LIN {X 0,Y 487.922,Z 777.858,A -85,B 0,C 180,E1 -6674.706,E2 -6674.706} C_VEL
LIN {X 0,Y 487.963,Z 774.749,A -85,B 0,C 180,E1 -6677.604,E2 -6677.604} C_VEL
LIN {X 0,Y 487.996,Z 771.009,A -85,B 0,C 180,E1 -6681.102,E2 -6681.102} C_VEL
LIN {X 0,Y 488.063,Z 768.175,A -85,B 0,C 180,E1 -6683.777,E2 -6683.777} C_VEL
LIN {X 0,Y 488.138,Z 765.028,A -85,B 0,C 180,E1 -6686.791,E2 -6686.791} C_VEL
LIN {X 0,Y 488.198,Z 761.474,A -85,B 0,C 180,E1 -6690.259,E2 -6690.259} C_VEL
LIN {X 0,Y 488.191,Z 760.678,A -85,B 0,C 180,E1 -6691.214,E2 -6691.214} C_VEL
LIN {X 0,Y 488.524,Z 760.636,A -85,B 0,C 180,E1 -6694.128,E2 -6694.128} C_VEL
LIN {X 0,Y 488.663,Z 760.617,A -85,B 0,C 180,E1 -6697.159,E2 -6697.159} C_VEL
LIN {X 0,Y 488.714,Z 760.606,A -85,B 0,C 180,E1 -6700.344,E2 -6700.344} C_VEL
LIN {X 0,Y 488.682,Z 760.613,A -85,B 0,C 180,E1 -6703.653,E2 -6703.653} C_VEL
LIN {X 0,Y 488.682,Z 760.609,A -85,B 0,C 180,E1 -6706.345,E2 -6706.345} C_VEL
LIN {X 0,Y 488.727,Z 760.607,A -85,B 0,C 180,E1 -6709.676,E2 -6709.676} C_VEL
LIN {X 0,Y 488.672,Z 760.612,A -85,B 0,C 180,E1 -6712.84,E2 -6712.84} C_VEL
LIN {X 0,Y 488.716,Z 760.608,A -85,B 0,C 180,E1 -6715.886,E2 -6715.886} C_VEL
LIN {X 0,Y 488.683,Z 760.609,A -85,B 0,C 180,E1 -6718.819,E2 -6718.819} C_VEL
LIN {X 0,Y 488.691,Z 760.607,A -85,B 0,C 180,E1 -6720.347,E2 -6720.347} C_VEL
LIN {X 0,Y 488.027,Z 760.693,A -85,B 0,C 180,E1 -6721.035,E2 -6721.035} C_VEL
LIN {X 0,Y 485.161,Z 761.049,A -85,B 0,C 180,E1 -6722.153,E2 -6722.153} C_VEL
LIN {X 0,Y 482.747,Z 761.35,A -85,B 0,C 180,E1 -6723.053,E2 -6723.053} C_VEL
LIN {X 0,Y 481.727,Z 761.48,A -85,B 0,C 180,E1 -6723.749,E2 -6723.749} C_VEL
LIN {X 0,Y 481.654,Z 761.487,A -85,B 0,C 180,E1 -6723.985,E2 -6723.985} C_VEL
LIN {X 0,Y 481.665,Z 761.483,A -85,B 0,C 180,E1 -6726.811,E2 -6726.811} C_VEL
LIN {X 0,Y 481.686,Z 761.486,A -85,B 0,C 180,E1 -6729.502,E2 -6729.502} C_VEL
LIN {X 0,Y 481.679,Z 761.484,A -85,B 0,C 180,E1 -6732.157,E2 -6732.157} C_VEL
LIN {X 0,Y 481.732,Z 761.474,A -85,B 0,C 180,E1 -6734.775,E2 -6734.775} C_VEL
LIN {X 0,Y 481.74,Z 761.476,A -85,B 0,C 180,E1 -6738.215,E2 -6738.215} C_VEL
LIN {X 0,Y 481.709,Z 761.481,A -85,B 0,C 180,E1 -6741.611,E2 -6741.611} C_VEL
LIN {X 0,Y 481.763,Z 761.475,A -85,B 0,C 180,E1 -6744.139,E2 -6744.139} C_VEL
LIN {X 0,Y 481.895,Z 761.455,A -85,B 0,C 180,E1 -6747.492,E2 -6747.492} C_VEL
LIN {X 0,Y 481.899,Z 761.461,A -85,B 0,C 180,E1 -6750,E2 -6750} C_VEL
LIN {X 0,Y 481.893,Z 761.456,A -85,B 0,C 180,E1 -6752.508,E2 -6752.508} C_VEL
LIN {X 0,Y 481.76,Z 761.474,A -85,B 0,C 180,E1 -6755.861,E2 -6755.861} C_VEL
LIN {X 0,Y 481.701,Z 761.483,A -85,B 0,C 180,E1 -6758.389,E2 -6758.389} C_VEL
LIN {X 0,Y 481.724,Z 761.477,A -85,B 0,C 180,E1 -6761.786,E2 -6761.786} C_VEL
LIN {X 0,Y 481.732,Z 761.474,A -85,B 0,C 180,E1 -6765.225,E2 -6765.225} C_VEL
LIN {X 0,Y 481.696,Z 761.482,A -85,B 0,C 180,E1 -6768.722,E2 -6768.722} C_VEL
LIN {X 0,Y 481.636,Z 761.486,A -85,B 0,C 180,E1 -6771.395,E2 -6771.395} C_VEL
LIN {X 0,Y 481.639,Z 761.489,A -85,B 0,C 180,E1 -6774.115,E2 -6774.115} C_VEL
LIN {X 0,Y 481.667,Z 761.483,A -85,B 0,C 180,E1 -6777.123,E2 -6777.123} C_VEL
LIN {X 0,Y 481.664,Z 761.483,A -85,B 0,C 180,E1 -6779.742,E2 -6779.742} C_VEL
LIN {X 0,Y 481.662,Z 761.49,A -85,B 0,C 180,E1 -6782.675,E2 -6782.675} C_VEL
LIN {X 0,Y 481.628,Z 761.488,A -85,B 0,C 180,E1 -6785.71,E2 -6785.71} C_VEL
LIN {X 0,Y 481.664,Z 761.489,A -85,B 0,C 180,E1 -6788.86,E2 -6788.86} C_VEL
LIN {X 0,Y 481.646,Z 761.486,A -85,B 0,C 180,E1 -6791.914,E2 -6791.914} C_VEL
LIN {X 0,Y 481.649,Z 761.489,A -85,B 0,C 180,E1 -6794.459,E2 -6794.459} C_VEL
LIN {X 0,Y 481.643,Z 761.486,A -85,B 0,C 180,E1 -6797.84,E2 -6797.84} C_VEL
LIN {X 0,Y 481.676,Z 761.486,A -85,B 0,C 180,E1 -6800.652,E2 -6800.652} C_VEL
LIN {X 0,Y 481.618,Z 761.492,A -85,B 0,C 180,E1 -6803.378,E2 -6803.378} C_VEL
LIN {X 0,Y 481.486,Z 761.51,A -85,B 0,C 180,E1 -6806.314,E2 -6806.314} C_VEL
LIN {X 0,Y 481.112,Z 761.559,A -85,B 0,C 180,E1 -6809.253,E2 -6809.253} C_VEL
LIN {X 0,Y 480.968,Z 761.685,A -85,B 0,C 180,E1 -6810.212,E2 -6810.212} C_VEL
LIN {X 0,Y 481.03,Z 764.86,A -85,B 0,C 180,E1 -6813.07,E2 -6813.07} C_VEL
LIN {X 0,Y 480.937,Z 767.926,A -85,B 0,C 180,E1 -6815.849,E2 -6815.849} C_VEL
LIN {X 0,Y 480.903,Z 770.923,A -85,B 0,C 180,E1 -6818.572,E2 -6818.572} C_VEL
LIN {X 0,Y 480.857,Z 773.831,A -85,B 0,C 180,E1 -6821.245,E2 -6821.245} C_VEL
LIN {X 0,Y 480.874,Z 777.672,A -85,B 0,C 180,E1 -6824.749,E2 -6824.749} C_VEL
LIN {X 0,Y 480.881,Z 778.156,A -85,B 0,C 180,E1 -6825.194,E2 -6825.194} C_VEL
LIN {X 0,Y 483.342,Z 790.593,A -85,B 0,C 180,E1 -6825.636,E2 -6825.636} C_VEL
LIN {X 0,Y 483.812,Z 796.114,A -85,B 0,C 180,E1 -6825.865,E2 -6825.865} C_VEL
LIN {X 0,Y 483.429,Z 808.116,A -85,B 0,C 180,E1 -6826.443,E2 -6826.443} C_VEL
LIN {X 0,Y 483.005,Z 820.229,A -85,B 0,C 180,E1 -6827.21,E2 -6827.21} C_VEL
LIN {X 0,Y 482.616,Z 831.531,A -85,B 0,C 180,E1 -6828.131,E2 -6828.131} C_VEL
LIN {X 0,Y 482.137,Z 840.94,A -85,B 0,C 180,E1 -6829.077,E2 -6829.077} C_VEL
LIN {X 0,Y 481.85,Z 849.541,A -85,B 0,C 180,E1 -6830.133,E2 -6830.133} C_VEL
LIN {X 0,Y 481.489,Z 857.935,A -85,B 0,C 180,E1 -6831.396,E2 -6831.396} C_VEL
LIN {X 0,Y 481.234,Z 863.639,A -85,B 0,C 180,E1 -6832.448,E2 -6832.448} C_VEL
LIN {X 0,Y 481.106,Z 869.017,A -85,B 0,C 180,E1 -6833.666,E2 -6833.666} C_VEL
LIN {X 0,Y 480.907,Z 873.547,A -85,B 0,C 180,E1 -6834.971,E2 -6834.971} C_VEL
LIN {X 0,Y 480.941,Z 875.835,A -85,B 0,C 180,E1 -6835.811,E2 -6835.811} C_VEL
LIN {X 0,Y 480.897,Z 877.707,A -85,B 0,C 180,E1 -6836.65,E2 -6836.65} C_VEL
LIN {X 0,Y 480.845,Z 879.143,A -85,B 0,C 180,E1 -6837.488,E2 -6837.488} C_VEL
LIN {X 0,Y 480.76,Z 880.779,A -85,B 0,C 180,E1 -6839.163,E2 -6839.163} C_VEL
LIN {X 0,Y 480.743,Z 881.028,A -85,B 0,C 180,E1 -6840.001,E2 -6840.001} C_VEL
LIN {X 0,Y 480.76,Z 880.847,A -85,B 0,C 180,E1 -6840.838,E2 -6840.838} C_VEL
LIN {X 0,Y 480.862,Z 879.314,A -85,B 0,C 180,E1 -6842.514,E2 -6842.514} C_VEL
LIN {X 0,Y 480.897,Z 877.961,A -85,B 0,C 180,E1 -6843.352,E2 -6843.352} C_VEL
LIN {X 0,Y 480.95,Z 875.11,A -85,B 0,C 180,E1 -6844.611,E2 -6844.611} C_VEL
LIN {X 0,Y 481.088,Z 871.224,A -85,B 0,C 180,E1 -6845.87,E2 -6845.87} C_VEL
LIN {X 0,Y 481.187,Z 866.185,A -85,B 0,C 180,E1 -6847.132,E2 -6847.132} C_VEL
LIN {X 0,Y 481.437,Z 859.82,A -85,B 0,C 180,E1 -6848.395,E2 -6848.395} C_VEL
LIN {X 0,Y 481.759,Z 851.905,A -85,B 0,C 180,E1 -6849.659,E2 -6849.659} C_VEL
LIN {X 0,Y 482.071,Z 843.809,A -85,B 0,C 180,E1 -6850.713,E2 -6850.713} C_VEL
LIN {X 0,Y 482.589,Z 833.83,A -85,B 0,C 180,E1 -6851.765,E2 -6851.765} C_VEL
LIN {X 0,Y 482.906,Z 822.414,A -85,B 0,C 180,E1 -6852.736,E2 -6852.736} C_VEL
LIN {X 0,Y 483.366,Z 811.702,A -85,B 0,C 180,E1 -6853.453,E2 -6853.453} C_VEL
LIN {X 0,Y 483.766,Z 799.439,A -85,B 0,C 180,E1 -6854.084,E2 -6854.084} C_VEL
LIN {X 0,Y 483.682,Z 793.011,A -85,B 0,C 180,E1 -6854.355,E2 -6854.355} C_VEL
LIN {X 0,Y 481.87,Z 782.956,A -85,B 0,C 180,E1 -6854.74,E2 -6854.74} C_VEL
LIN {X 0,Y 480.939,Z 778.913,A -85,B 0,C 180,E1 -6854.899,E2 -6854.899} C_VEL
LIN {X 0,Y 480.94,Z 775.326,A -85,B 0,C 180,E1 -6858.222,E2 -6858.222} C_VEL
LIN {X 0,Y 480.955,Z 771.748,A -85,B 0,C 180,E1 -6861.428,E2 -6861.428} C_VEL
LIN {X 0,Y 480.98,Z 768.696,A -85,B 0,C 180,E1 -6864.151,E2 -6864.151} C_VEL
LIN {X 0,Y 481.015,Z 765.283,A -85,B 0,C 180,E1 -6866.968,E2 -6866.968} C_VEL
LIN {X 0,Y 480.974,Z 761.647,A -85,B 0,C 180,E1 -6869.79,E2 -6869.79} C_VEL
LIN {X 0,Y 481.36,Z 761.528,A -85,B 0,C 180,E1 -6872.699,E2 -6872.699} C_VEL
LIN {X 0,Y 481.595,Z 761.495,A -85,B 0,C 180,E1 -6875.714,E2 -6875.714} C_VEL
LIN {X 0,Y 481.675,Z 761.487,A -85,B 0,C 180,E1 -6878.859,E2 -6878.859} C_VEL
LIN {X 0,Y 481.651,Z 761.486,A -85,B 0,C 180,E1 -6881.912,E2 -6881.912} C_VEL
LIN {X 0,Y 481.664,Z 761.486,A -85,B 0,C 180,E1 -6884.458,E2 -6884.458} C_VEL
LIN {X 0,Y 481.652,Z 761.487,A -85,B 0,C 180,E1 -6887.84,E2 -6887.84} C_VEL
LIN {X 0,Y 481.701,Z 761.516,A -85,B 0,C 180,E1 -6889.801,E2 -6889.801} C_VEL
LIN {X 0,Y 482.913,Z 768.412,A -85,B 0,C 180,E1 -6892.774,E2 -6892.774} C_VEL
LIN {X 0,Y 483.335,Z 772.686,A -85,B 0,C 180,E1 -6894.517,E2 -6894.517} C_VEL
LIN {X 0,Y 482.962,Z 780.236,A -85,B 0,C 180,E1 -6897.424,E2 -6897.424} C_VEL
LIN {X 0,Y 482.594,Z 788.032,A -85,B 0,C 180,E1 -6900.321,E2 -6900.321} C_VEL
LIN {X 0,Y 482.239,Z 795.887,A -85,B 0,C 180,E1 -6903.142,E2 -6903.142} C_VEL
LIN {X 0,Y 481.961,Z 803.794,A -85,B 0,C 180,E1 -6905.902,E2 -6905.902} C_VEL
LIN {X 0,Y 481.677,Z 813.021,A -85,B 0,C 180,E1 -6909.037,E2 -6909.037} C_VEL
LIN {X 0,Y 481.429,Z 822.408,A -85,B 0,C 180,E1 -6912.148,E2 -6912.148} C_VEL
LIN {X 0,Y 481.282,Z 831.603,A -85,B 0,C 180,E1 -6915.072,E2 -6915.072} C_VEL
LIN {X 0,Y 483.425,Z 845.293,A -85,B 0,C 180,E1 -6915.49,E2 -6915.49} C_VEL
LIN {X 0,Y 483.816,Z 849.512,A -85,B 0,C 180,E1 -6915.649,E2 -6915.649} C_VEL
LIN {X 0,Y 483.512,Z 861.696,A -85,B 0,C 180,E1 -6916.177,E2 -6916.177} C_VEL
LIN {X 0,Y 483.027,Z 873.992,A -85,B 0,C 180,E1 -6916.891,E2 -6916.891} C_VEL
LIN {X 0,Y 482.617,Z 884.929,A -85,B 0,C 180,E1 -6917.703,E2 -6917.703} C_VEL
LIN {X 0,Y 482.23,Z 895.247,A -85,B 0,C 180,E1 -6918.653,E2 -6918.653} C_VEL
LIN {X 0,Y 481.821,Z 904.529,A -85,B 0,C 180,E1 -6919.707,E2 -6919.707} C_VEL
LIN {X 0,Y 481.453,Z 913.564,A -85,B 0,C 180,E1 -6920.972,E2 -6920.972} C_VEL
LIN {X 0,Y 481.18,Z 920.842,A -85,B 0,C 180,E1 -6922.235,E2 -6922.235} C_VEL
LIN {X 0,Y 481.025,Z 926.557,A -85,B 0,C 180,E1 -6923.473,E2 -6923.473} C_VEL
LIN {X 0,Y 480.979,Z 930.536,A -85,B 0,C 180,E1 -6924.55,E2 -6924.55} C_VEL
LIN {X 0,Y 480.85,Z 934.181,A -85,B 0,C 180,E1 -6925.809,E2 -6925.809} C_VEL
LIN {X 0,Y 480.892,Z 936.066,A -85,B 0,C 180,E1 -6926.649,E2 -6926.649} C_VEL
LIN {X 0,Y 480.819,Z 938.478,A -85,B 0,C 180,E1 -6928.325,E2 -6928.325} C_VEL
LIN {X 0,Y 480.76,Z 939.086,A -85,B 0,C 180,E1 -6929.162,E2 -6929.162} C_VEL
LIN {X 0,Y 480.743,Z 939.297,A -85,B 0,C 180,E1 -6930,E2 -6930} C_VEL
LIN {X 0,Y 480.819,Z 938.457,A -85,B 0,C 180,E1 -6931.675,E2 -6931.675} C_VEL
LIN {X 0,Y 480.804,Z 937.443,A -85,B 0,C 180,E1 -6932.513,E2 -6932.513} C_VEL
LIN {X 0,Y 480.892,Z 936.018,A -85,B 0,C 180,E1 -6933.351,E2 -6933.351} C_VEL
LIN {X 0,Y 480.854,Z 933.023,A -85,B 0,C 180,E1 -6934.611,E2 -6934.611} C_VEL
LIN {X 0,Y 481.003,Z 928.98,A -85,B 0,C 180,E1 -6935.87,E2 -6935.87} C_VEL
LIN {X 0,Y 481.115,Z 922.75,A -85,B 0,C 180,E1 -6937.344,E2 -6937.344} C_VEL
LIN {X 0,Y 481.368,Z 915.951,A -85,B 0,C 180,E1 -6938.607,E2 -6938.607} C_VEL
LIN {X 0,Y 481.668,Z 907.498,A -85,B 0,C 180,E1 -6939.872,E2 -6939.872} C_VEL
LIN {X 0,Y 481.993,Z 898.816,A -85,B 0,C 180,E1 -6940.927,E2 -6940.927} C_VEL
LIN {X 0,Y 482.463,Z 888.126,A -85,B 0,C 180,E1 -6941.981,E2 -6941.981} C_VEL
LIN {X 0,Y 482.864,Z 876.533,A -85,B 0,C 180,E1 -6942.899,E2 -6942.899} C_VEL
LIN {X 0,Y 483.32,Z 863.934,A -85,B 0,C 180,E1 -6943.668,E2 -6943.668} C_VEL
LIN {X 0,Y 483.741,Z 851.423,A -85,B 0,C 180,E1 -6944.245,E2 -6944.245} C_VEL
LIN {X 0,Y 483.593,Z 846.689,A -85,B 0,C 180,E1 -6944.424,E2 -6944.424} C_VEL
LIN {X 0,Y 481.609,Z 833.971,A -85,B 0,C 180,E1 -6944.846,E2 -6944.846} C_VEL
LIN {X 0,Y 481.222,Z 830.609,A -85,B 0,C 180,E1 -6944.943,E2 -6944.943} C_VEL
LIN {X 0,Y 481.439,Z 819.625,A -85,B 0,C 180,E1 -6948.401,E2 -6948.401} C_VEL
LIN {X 0,Y 481.591,Z 810.298,A -85,B 0,C 180,E1 -6951.397,E2 -6951.397} C_VEL
LIN {X 0,Y 481.791,Z 802.077,A -85,B 0,C 180,E1 -6954.107,E2 -6954.107} C_VEL
LIN {X 0,Y 482.069,Z 793.079,A -85,B 0,C 180,E1 -6957.213,E2 -6957.213} C_VEL
LIN {X 0,Y 482.387,Z 784.985,A -85,B 0,C 180,E1 -6960.175,E2 -6960.175} C_VEL
LIN {X 0,Y 482.87,Z 777.717,A -85,B 0,C 180,E1 -6963.079,E2 -6963.079} C_VEL
LIN {X 0,Y 483.209,Z 772.182,A -85,B 0,C 180,E1 -6965.576,E2 -6965.576} C_VEL
LIN {X 0,Y 483.08,Z 769.718,A -85,B 0,C 180,E1 -6966.854,E2 -6966.854} C_VEL
LIN {X 0,Y 482.367,Z 765.546,A -85,B 0,C 180,E1 -6969.447,E2 -6969.447} C_VEL
LIN {X 0,Y 481.876,Z 762.588,A -85,B 0,C 180,E1 -6971.942,E2 -6971.942} C_VEL
LIN {X 0,Y 481.644,Z 761.493,A -85,B 0,C 180,E1 -6973.3,E2 -6973.3} C_VEL
LIN {X 0,Y 481.662,Z 761.49,A -85,B 0,C 180,E1 -6975.641,E2 -6975.641} C_VEL
LIN {X 0,Y 481.652,Z 761.492,A -85,B 0,C 180,E1 -6978.957,E2 -6978.957} C_VEL
LIN {X 0,Y 481.654,Z 761.491,A -85,B 0,C 180,E1 -6981.993,E2 -6981.993} C_VEL
LIN {X 0,Y 481.62,Z 761.496,A -85,B 0,C 180,E1 -6983.378,E2 -6983.378} C_VEL
LIN {X 0,Y 481.674,Z 763.122,A -85,B 0,C 180,E1 -6986.326,E2 -6986.326} C_VEL
LIN {X 0,Y 481.482,Z 765.201,A -85,B 0,C 180,E1 -6989.277,E2 -6989.277} C_VEL
LIN {X 0,Y 481.323,Z 767.426,A -85,B 0,C 180,E1 -6992.144,E2 -6992.144} C_VEL
LIN {X 0,Y 481.214,Z 769.746,A -85,B 0,C 180,E1 -6994.941,E2 -6994.941} C_VEL
LIN {X 0,Y 481.126,Z 772.136,A -85,B 0,C 180,E1 -6997.678,E2 -6997.678} C_VEL
LIN {X 0,Y 481.035,Z 774.58,A -85,B 0,C 180,E1 -7000.364,E2 -7000.364} C_VEL
LIN {X 0,Y 480.94,Z 777.081,A -85,B 0,C 180,E1 -7003.006,E2 -7003.006} C_VEL
LIN {X 0,Y 480.978,Z 779.353,A -85,B 0,C 180,E1 -7005.215,E2 -7005.215} C_VEL
LIN {X 0,Y 483.165,Z 789.409,A -85,B 0,C 180,E1 -7005.575,E2 -7005.575} C_VEL
LIN {X 0,Y 483.895,Z 795.128,A -85,B 0,C 180,E1 -7005.812,E2 -7005.812} C_VEL
LIN {X 0,Y 483.558,Z 806.516,A -85,B 0,C 180,E1 -7006.338,E2 -7006.338} C_VEL
LIN {X 0,Y 483.151,Z 818.394,A -85,B 0,C 180,E1 -7007.058,E2 -7007.058} C_VEL
LIN {X 0,Y 482.773,Z 829.526,A -85,B 0,C 180,E1 -7007.92,E2 -7007.92} C_VEL
LIN {X 0,Y 482.307,Z 839.336,A -85,B 0,C 180,E1 -7008.867,E2 -7008.867} C_VEL
LIN {X 0,Y 481.944,Z 848.244,A -85,B 0,C 180,E1 -7009.921,E2 -7009.921} C_VEL
LIN {X 0,Y 481.554,Z 856.932,A -85,B 0,C 180,E1 -7011.184,E2 -7011.184} C_VEL
LIN {X 0,Y 481.253,Z 863.851,A -85,B 0,C 180,E1 -7012.447,E2 -7012.447} C_VEL
LIN {X 0,Y 481.146,Z 869.127,A -85,B 0,C 180,E1 -7013.647,E2 -7013.647} C_VEL
LIN {X 0,Y 480.91,Z 873.698,A -85,B 0,C 180,E1 -7014.969,E2 -7014.969} C_VEL
LIN {X 0,Y 480.961,Z 875.974,A -85,B 0,C 180,E1 -7015.809,E2 -7015.809} C_VEL
LIN {X 0,Y 480.898,Z 877.833,A -85,B 0,C 180,E1 -7016.648,E2 -7016.648} C_VEL
LIN {X 0,Y 480.862,Z 879.237,A -85,B 0,C 180,E1 -7017.486,E2 -7017.486} C_VEL
LIN {X 0,Y 480.76,Z 880.838,A -85,B 0,C 180,E1 -7019.162,E2 -7019.162} C_VEL
LIN {X 0,Y 480.743,Z 881.064,A -85,B 0,C 180,E1 -7019.999,E2 -7019.999} C_VEL
LIN {X 0,Y 480.76,Z 880.87,A -85,B 0,C 180,E1 -7020.837,E2 -7020.837} C_VEL
LIN {X 0,Y 480.82,Z 880.276,A -85,B 0,C 180,E1 -7021.674,E2 -7021.674} C_VEL
LIN {X 0,Y 480.897,Z 877.926,A -85,B 0,C 180,E1 -7023.35,E2 -7023.35} C_VEL
LIN {X 0,Y 480.917,Z 875.044,A -85,B 0,C 180,E1 -7024.609,E2 -7024.609} C_VEL
LIN {X 0,Y 481.081,Z 871.13,A -85,B 0,C 180,E1 -7025.868,E2 -7025.868} C_VEL
LIN {X 0,Y 481.176,Z 866.086,A -85,B 0,C 180,E1 -7027.131,E2 -7027.131} C_VEL
LIN {X 0,Y 481.437,Z 859.72,A -85,B 0,C 180,E1 -7028.393,E2 -7028.393} C_VEL
LIN {X 0,Y 481.765,Z 851.763,A -85,B 0,C 180,E1 -7029.657,E2 -7029.657} C_VEL
LIN {X 0,Y 482.062,Z 843.642,A -85,B 0,C 180,E1 -7030.712,E2 -7030.712} C_VEL
LIN {X 0,Y 482.567,Z 833.73,A -85,B 0,C 180,E1 -7031.764,E2 -7031.764} C_VEL
LIN {X 0,Y 482.928,Z 823.956,A -85,B 0,C 180,E1 -7032.608,E2 -7032.608} C_VEL
LIN {X 0,Y 483.281,Z 813.302,A -85,B 0,C 180,E1 -7033.35,E2 -7033.35} C_VEL
LIN {X 0,Y 483.716,Z 800.661,A -85,B 0,C 180,E1 -7034.031,E2 -7034.031} C_VEL
LIN {X 0,Y 483.677,Z 792.833,A -85,B 0,C 180,E1 -7034.367,E2 -7034.367} C_VEL
LIN {X 0,Y 481.717,Z 782.039,A -85,B 0,C 180,E1 -7034.779,E2 -7034.779} C_VEL
LIN {X 0,Y 480.87,Z 778.199,A -85,B 0,C 180,E1 -7034.926,E2 -7034.926} C_VEL
LIN {X 0,Y 480.891,Z 774.679,A -85,B 0,C 180,E1 -7038.204,E2 -7038.204} C_VEL
LIN {X 0,Y 480.936,Z 771.266,A -85,B 0,C 180,E1 -7041.427,E2 -7041.427} C_VEL
LIN {X 0,Y 480.98,Z 768.41,A -85,B 0,C 180,E1 -7044.149,E2 -7044.149} C_VEL
LIN {X 0,Y 481.053,Z 765.488,A -85,B 0,C 180,E1 -7046.977,E2 -7046.977} C_VEL
LIN {X 0,Y 481.136,Z 761.903,A -85,B 0,C 180,E1 -7050.478,E2 -7050.478} C_VEL
LIN {X 0,Y 481.213,Z 761.547,A -85,B 0,C 180,E1 -7051.719,E2 -7051.719} C_VEL
LIN {X 0,Y 481.534,Z 761.506,A -85,B 0,C 180,E1 -7054.694,E2 -7054.694} C_VEL
LIN {X 0,Y 481.62,Z 761.491,A -85,B 0,C 180,E1 -7057.797,E2 -7057.797} C_VEL
LIN {X 0,Y 481.658,Z 761.486,A -85,B 0,C 180,E1 -7060.646,E2 -7060.646} C_VEL
LIN {X 0,Y 481.634,Z 761.492,A -85,B 0,C 180,E1 -7063.299,E2 -7063.299} C_VEL
LIN {X 0,Y 481.653,Z 761.488,A -85,B 0,C 180,E1 -7065.64,E2 -7065.64} C_VEL
LIN {X 0,Y 481.65,Z 761.488,A -85,B 0,C 180,E1 -7068.957,E2 -7068.957} C_VEL
LIN {X 0,Y 481.648,Z 761.488,A -85,B 0,C 180,E1 -7071.992,E2 -7071.992} C_VEL
LIN {X 0,Y 481.677,Z 761.488,A -85,B 0,C 180,E1 -7075.317,E2 -7075.317} C_VEL
LIN {X 0,Y 481.636,Z 761.487,A -85,B 0,C 180,E1 -7078.311,E2 -7078.311} C_VEL
LIN {X 0,Y 481.667,Z 761.486,A -85,B 0,C 180,E1 -7081.216,E2 -7081.216} C_VEL
LIN {X 0,Y 481.654,Z 761.487,A -85,B 0,C 180,E1 -7083.985,E2 -7083.985} C_VEL
LIN {X 0,Y 481.01,Z 761.571,A -85,B 0,C 180,E1 -7084.683,E2 -7084.683} C_VEL
LIN {X 0,Y 478.154,Z 761.929,A -85,B 0,C 180,E1 -7085.816,E2 -7085.816} C_VEL
LIN {X 0,Y 475.717,Z 762.23,A -85,B 0,C 180,E1 -7086.73,E2 -7086.73} C_VEL
LIN {X 0,Y 474.663,Z 762.36,A -85,B 0,C 180,E1 -7087.436,E2 -7087.436} C_VEL
LIN {X 0,Y 474.573,Z 762.368,A -85,B 0,C 180,E1 -7087.675,E2 -7087.675} C_VEL
LIN {X 0,Y 474.644,Z 762.36,A -85,B 0,C 180,E1 -7090.089,E2 -7090.089} C_VEL
LIN {X 0,Y 474.625,Z 762.36,A -85,B 0,C 180,E1 -7092.773,E2 -7092.773} C_VEL
LIN {X 0,Y 474.636,Z 762.362,A -85,B 0,C 180,E1 -7095.421,E2 -7095.421} C_VEL
LIN {X 0,Y 474.694,Z 762.355,A -85,B 0,C 180,E1 -7098.037,E2 -7098.037} C_VEL
LIN {X 0,Y 474.685,Z 762.355,A -85,B 0,C 180,E1 -7101.486,E2 -7101.486} C_VEL
LIN {X 0,Y 474.726,Z 762.353,A -85,B 0,C 180,E1 -7104.052,E2 -7104.052} C_VEL
LIN {X 0,Y 474.86,Z 762.331,A -85,B 0,C 180,E1 -7107.455,E2 -7107.455} C_VEL
LIN {X 0,Y 474.868,Z 762.337,A -85,B 0,C 180,E1 -7110,E2 -7110} C_VEL
LIN {X 0,Y 474.858,Z 762.332,A -85,B 0,C 180,E1 -7112.545,E2 -7112.545} C_VEL
LIN {X 0,Y 474.724,Z 762.352,A -85,B 0,C 180,E1 -7115.948,E2 -7115.948} C_VEL
LIN {X 0,Y 474.65,Z 762.36,A -85,B 0,C 180,E1 -7118.515,E2 -7118.515} C_VEL
LIN {X 0,Y 474.682,Z 762.356,A -85,B 0,C 180,E1 -7121.963,E2 -7121.963} C_VEL
LIN {X 0,Y 474.689,Z 762.351,A -85,B 0,C 180,E1 -7125.456,E2 -7125.456} C_VEL
LIN {X 0,Y 474.651,Z 762.357,A -85,B 0,C 180,E1 -7129.011,E2 -7129.011} C_VEL
LIN {X 0,Y 474.579,Z 762.366,A -85,B 0,C 180,E1 -7131.729,E2 -7131.729} C_VEL
LIN {X 0,Y 474.617,Z 762.368,A -85,B 0,C 180,E1 -7134.495,E2 -7134.495} C_VEL
LIN {X 0,Y 474.628,Z 762.36,A -85,B 0,C 180,E1 -7137.325,E2 -7137.325} C_VEL
LIN {X 0,Y 474.594,Z 762.367,A -85,B 0,C 180,E1 -7140.231,E2 -7140.231} C_VEL
LIN {X 0,Y 474.617,Z 762.362,A -85,B 0,C 180,E1 -7143.222,E2 -7143.222} C_VEL
LIN {X 0,Y 474.581,Z 762.369,A -85,B 0,C 180,E1 -7146.324,E2 -7146.324} C_VEL
LIN {X 0,Y 474.611,Z 762.362,A -85,B 0,C 180,E1 -7149.647,E2 -7149.647} C_VEL
LIN {X 0,Y 474.608,Z 762.368,A -85,B 0,C 180,E1 -7152.935,E2 -7152.935} C_VEL
LIN {X 0,Y 474.601,Z 762.364,A -85,B 0,C 180,E1 -7155.896,E2 -7155.896} C_VEL
LIN {X 0,Y 474.623,Z 762.366,A -85,B 0,C 180,E1 -7159.042,E2 -7159.042} C_VEL
LIN {X 0,Y 474.605,Z 762.363,A -85,B 0,C 180,E1 -7161.705,E2 -7161.705} C_VEL
LIN {X 0,Y 474.549,Z 762.373,A -85,B 0,C 180,E1 -7164.721,E2 -7164.721} C_VEL
LIN {X 0,Y 474.296,Z 762.408,A -85,B 0,C 180,E1 -7167.763,E2 -7167.763} C_VEL
LIN {X 0,Y 473.984,Z 762.447,A -85,B 0,C 180,E1 -7169.727,E2 -7169.727} C_VEL
LIN {X 0,Y 473.907,Z 763.208,A -85,B 0,C 180,E1 -7171.041,E2 -7171.041} C_VEL
LIN {X 0,Y 473.933,Z 766.021,A -85,B 0,C 180,E1 -7173.586,E2 -7173.586} C_VEL
LIN {X 0,Y 473.873,Z 769.596,A -85,B 0,C 180,E1 -7176.857,E2 -7176.857} C_VEL
LIN {X 0,Y 473.81,Z 773.121,A -85,B 0,C 180,E1 -7180.054,E2 -7180.054} C_VEL
LIN {X 0,Y 473.755,Z 776.046,A -85,B 0,C 180,E1 -7182.742,E2 -7182.742} C_VEL
LIN {X 0,Y 473.82,Z 778.588,A -85,B 0,C 180,E1 -7184.98,E2 -7184.98} C_VEL
LIN {X 0,Y 476.324,Z 790.746,A -85,B 0,C 180,E1 -7185.422,E2 -7185.422} C_VEL
LIN {X 0,Y 476.922,Z 796.22,A -85,B 0,C 180,E1 -7185.657,E2 -7185.657} C_VEL
LIN {X 0,Y 476.527,Z 808.264,A -85,B 0,C 180,E1 -7186.243,E2 -7186.243} C_VEL
LIN {X 0,Y 476.072,Z 819.969,A -85,B 0,C 180,E1 -7186.989,E2 -7186.989} C_VEL
LIN {X 0,Y 475.709,Z 830.603,A -85,B 0,C 180,E1 -7187.848,E2 -7187.848} C_VEL
LIN {X 0,Y 475.172,Z 841.186,A -85,B 0,C 180,E1 -7188.915,E2 -7188.915} C_VEL
LIN {X 0,Y 474.859,Z 849.815,A -85,B 0,C 180,E1 -7189.986,E2 -7189.986} C_VEL
LIN {X 0,Y 474.461,Z 858.242,A -85,B 0,C 180,E1 -7191.268,E2 -7191.268} C_VEL
LIN {X 0,Y 474.192,Z 863.966,A -85,B 0,C 180,E1 -7192.335,E2 -7192.335} C_VEL
LIN {X 0,Y 474.042,Z 869.687,A -85,B 0,C 180,E1 -7193.657,E2 -7193.657} C_VEL
LIN {X 0,Y 473.847,Z 873.915,A -85,B 0,C 180,E1 -7194.895,E2 -7194.895} C_VEL
LIN {X 0,Y 473.871,Z 876.212,A -85,B 0,C 180,E1 -7195.748,E2 -7195.748} C_VEL
LIN {X 0,Y 473.828,Z 878.096,A -85,B 0,C 180,E1 -7196.6,E2 -7196.6} C_VEL
LIN {X 0,Y 473.761,Z 879.542,A -85,B 0,C 180,E1 -7197.45,E2 -7197.45} C_VEL
LIN {X 0,Y 473.753,Z 880.554,A -85,B 0,C 180,E1 -7198.301,E2 -7198.301} C_VEL
LIN {X 0,Y 473.669,Z 881.444,A -85,B 0,C 180,E1 -7200.001,E2 -7200.001} C_VEL
LIN {X 0,Y 473.689,Z 881.265,A -85,B 0,C 180,E1 -7200.851,E2 -7200.851} C_VEL
LIN {X 0,Y 473.79,Z 879.734,A -85,B 0,C 180,E1 -7202.551,E2 -7202.551} C_VEL
LIN {X 0,Y 473.83,Z 878.377,A -85,B 0,C 180,E1 -7203.402,E2 -7203.402} C_VEL
LIN {X 0,Y 473.878,Z 875.521,A -85,B 0,C 180,E1 -7204.68,E2 -7204.68} C_VEL
LIN {X 0,Y 474.04,Z 871.623,A -85,B 0,C 180,E1 -7205.958,E2 -7205.958} C_VEL
LIN {X 0,Y 474.139,Z 866.567,A -85,B 0,C 180,E1 -7207.239,E2 -7207.239} C_VEL
LIN {X 0,Y 474.409,Z 860.183,A -85,B 0,C 180,E1 -7208.52,E2 -7208.52} C_VEL
LIN {X 0,Y 474.784,Z 852.243,A -85,B 0,C 180,E1 -7209.802,E2 -7209.802} C_VEL
LIN {X 0,Y 475.103,Z 844.121,A -85,B 0,C 180,E1 -7210.872,E2 -7210.872} C_VEL
LIN {X 0,Y 475.654,Z 834.097,A -85,B 0,C 180,E1 -7211.939,E2 -7211.939} C_VEL
LIN {X 0,Y 475.973,Z 823.027,A -85,B 0,C 180,E1 -7212.894,E2 -7212.894} C_VEL
LIN {X 0,Y 476.456,Z 811.87,A -85,B 0,C 180,E1 -7213.652,E2 -7213.652} C_VEL
LIN {X 0,Y 476.893,Z 799.555,A -85,B 0,C 180,E1 -7214.292,E2 -7214.292} C_VEL
LIN {X 0,Y 476.856,Z 794.471,A -85,B 0,C 180,E1 -7214.511,E2 -7214.511} C_VEL
LIN {X 0,Y 475.033,Z 784.289,A -85,B 0,C 180,E1 -7214.92,E2 -7214.92} C_VEL
LIN {X 0,Y 473.896,Z 779.417,A -85,B 0,C 180,E1 -7215.101,E2 -7215.101} C_VEL
LIN {X 0,Y 473.886,Z 775.893,A -85,B 0,C 180,E1 -7218.348,E2 -7218.348} C_VEL
LIN {X 0,Y 473.89,Z 772.101,A -85,B 0,C 180,E1 -7221.763,E2 -7221.763} C_VEL
LIN {X 0,Y 473.921,Z 768.987,A -85,B 0,C 180,E1 -7224.534,E2 -7224.534} C_VEL
LIN {X 0,Y 473.94,Z 765.585,A -85,B 0,C 180,E1 -7227.368,E2 -7227.368} C_VEL
LIN {X 0,Y 473.903,Z 763.035,A -85,B 0,C 180,E1 -7229.301,E2 -7229.301} C_VEL
LIN {X 0,Y 474.046,Z 762.44,A -85,B 0,C 180,E1 -7230.696,E2 -7230.696} C_VEL
LIN {X 0,Y 474.36,Z 762.4,A -85,B 0,C 180,E1 -7233.243,E2 -7233.243} C_VEL
LIN {X 0,Y 474.554,Z 762.375,A -85,B 0,C 180,E1 -7235.458,E2 -7235.458} C_VEL
LIN {X 0,Y 474.615,Z 762.364,A -85,B 0,C 180,E1 -7238.458,E2 -7238.458} C_VEL
LIN {X 0,Y 474.619,Z 762.363,A -85,B 0,C 180,E1 -7241.786,E2 -7241.786} C_VEL
LIN {X 0,Y 474.626,Z 762.366,A -85,B 0,C 180,E1 -7245.297,E2 -7245.297} C_VEL
LIN {X 0,Y 474.625,Z 762.363,A -85,B 0,C 180,E1 -7248.215,E2 -7248.215} C_VEL
LIN {X 0,Y 474.655,Z 762.438,A -85,B 0,C 180,E1 -7249.539,E2 -7249.539} C_VEL
LIN {X 0,Y 475.946,Z 769.75,A -85,B 0,C 180,E1 -7252.741,E2 -7252.741} C_VEL
LIN {X 0,Y 476.349,Z 773.344,A -85,B 0,C 180,E1 -7254.24,E2 -7254.24} C_VEL
LIN {X 0,Y 476.074,Z 780.092,A -85,B 0,C 180,E1 -7256.892,E2 -7256.892} C_VEL
LIN {X 0,Y 475.63,Z 787.881,A -85,B 0,C 180,E1 -7259.842,E2 -7259.842} C_VEL
LIN {X 0,Y 475.281,Z 795.713,A -85,B 0,C 180,E1 -7262.716,E2 -7262.716} C_VEL
LIN {X 0,Y 474.911,Z 804.912,A -85,B 0,C 180,E1 -7265.986,E2 -7265.986} C_VEL
LIN {X 0,Y 474.594,Z 814.15,A -85,B 0,C 180,E1 -7269.182,E2 -7269.182} C_VEL
LIN {X 0,Y 474.36,Z 823.446,A -85,B 0,C 180,E1 -7272.319,E2 -7272.319} C_VEL
LIN {X 0,Y 474.186,Z 831.04,A -85,B 0,C 180,E1 -7274.844,E2 -7274.844} C_VEL
LIN {X 0,Y 476.317,Z 845.099,A -85,B 0,C 180,E1 -7275.282,E2 -7275.282} C_VEL
LIN {X 0,Y 476.896,Z 850.372,A -85,B 0,C 180,E1 -7275.491,E2 -7275.491} C_VEL
LIN {X 0,Y 476.564,Z 862.146,A -85,B 0,C 180,E1 -7276.026,E2 -7276.026} C_VEL
LIN {X 0,Y 476.069,Z 873.452,A -85,B 0,C 180,E1 -7276.696,E2 -7276.696} C_VEL
LIN {X 0,Y 475.682,Z 883.928,A -85,B 0,C 180,E1 -7277.481,E2 -7277.481} C_VEL
LIN {X 0,Y 475.24,Z 894.739,A -85,B 0,C 180,E1 -7278.484,E2 -7278.484} C_VEL
LIN {X 0,Y 474.797,Z 904.044,A -85,B 0,C 180,E1 -7279.553,E2 -7279.553} C_VEL
LIN {X 0,Y 474.406,Z 913.092,A -85,B 0,C 180,E1 -7280.836,E2 -7280.836} C_VEL
LIN {X 0,Y 474.105,Z 920.384,A -85,B 0,C 180,E1 -7282.119,E2 -7282.119} C_VEL
LIN {X 0,Y 473.92,Z 926.622,A -85,B 0,C 180,E1 -7283.506,E2 -7283.506} C_VEL
LIN {X 0,Y 473.843,Z 931.432,A -85,B 0,C 180,E1 -7284.894,E2 -7284.894} C_VEL
LIN {X 0,Y 473.754,Z 933.752,A -85,B 0,C 180,E1 -7285.746,E2 -7285.746} C_VEL
LIN {X 0,Y 473.818,Z 935.642,A -85,B 0,C 180,E1 -7286.599,E2 -7286.599} C_VEL
LIN {X 0,Y 473.751,Z 938.057,A -85,B 0,C 180,E1 -7288.3,E2 -7288.3} C_VEL
LIN {X 0,Y 473.689,Z 938.662,A -85,B 0,C 180,E1 -7289.15,E2 -7289.15} C_VEL
LIN {X 0,Y 473.67,Z 938.87,A -85,B 0,C 180,E1 -7290,E2 -7290} C_VEL
LIN {X 0,Y 473.751,Z 938.022,A -85,B 0,C 180,E1 -7291.7,E2 -7291.7} C_VEL
LIN {X 0,Y 473.724,Z 936.995,A -85,B 0,C 180,E1 -7292.551,E2 -7292.551} C_VEL
LIN {X 0,Y 473.818,Z 935.561,A -85,B 0,C 180,E1 -7293.401,E2 -7293.401} C_VEL
LIN {X 0,Y 473.776,Z 932.548,A -85,B 0,C 180,E1 -7294.68,E2 -7294.68} C_VEL
LIN {X 0,Y 473.905,Z 928.481,A -85,B 0,C 180,E1 -7295.959,E2 -7295.959} C_VEL
LIN {X 0,Y 474.03,Z 922.22,A -85,B 0,C 180,E1 -7297.454,E2 -7297.454} C_VEL
LIN {X 0,Y 474.317,Z 915.388,A -85,B 0,C 180,E1 -7298.736,E2 -7298.736} C_VEL
LIN {X 0,Y 474.604,Z 906.894,A -85,B 0,C 180,E1 -7300.02,E2 -7300.02} C_VEL
LIN {X 0,Y 474.985,Z 898.171,A -85,B 0,C 180,E1 -7301.09,E2 -7301.09} C_VEL
LIN {X 0,Y 475.475,Z 887.589,A -85,B 0,C 180,E1 -7302.146,E2 -7302.146} C_VEL
LIN {X 0,Y 475.894,Z 875.798,A -85,B 0,C 180,E1 -7303.091,E2 -7303.091} C_VEL
LIN {X 0,Y 476.388,Z 863.157,A -85,B 0,C 180,E1 -7303.871,E2 -7303.871} C_VEL
LIN {X 0,Y 476.842,Z 850.619,A -85,B 0,C 180,E1 -7304.456,E2 -7304.456} C_VEL
LIN {X 0,Y 476.061,Z 843.865,A -85,B 0,C 180,E1 -7304.726,E2 -7304.726} C_VEL
LIN {X 0,Y 474.204,Z 830.784,A -85,B 0,C 180,E1 -7305.128,E2 -7305.128} C_VEL
LIN {X 0,Y 474.178,Z 830.142,A -85,B 0,C 180,E1 -7305.143,E2 -7305.143} C_VEL
LIN {X 0,Y 474.357,Z 819.633,A -85,B 0,C 180,E1 -7308.519,E2 -7308.519} C_VEL
LIN {X 0,Y 474.544,Z 809.831,A -85,B 0,C 180,E1 -7311.731,E2 -7311.731} C_VEL
LIN {X 0,Y 474.769,Z 801.683,A -85,B 0,C 180,E1 -7314.487,E2 -7314.487} C_VEL
LIN {X 0,Y 475.085,Z 792.396,A -85,B 0,C 180,E1 -7317.79,E2 -7317.79} C_VEL
LIN {X 0,Y 475.549,Z 783.616,A -85,B 0,C 180,E1 -7321.148,E2 -7321.148} C_VEL
LIN {X 0,Y 476.077,Z 776.383,A -85,B 0,C 180,E1 -7324.239,E2 -7324.239} C_VEL
LIN {X 0,Y 476.26,Z 772.403,A -85,B 0,C 180,E1 -7326.176,E2 -7326.176} C_VEL
LIN {X 0,Y 475.704,Z 768.524,A -85,B 0,C 180,E1 -7328.462,E2 -7328.462} C_VEL
LIN {X 0,Y 475.136,Z 765.12,A -85,B 0,C 180,E1 -7331.029,E2 -7331.029} C_VEL
LIN {X 0,Y 474.706,Z 762.911,A -85,B 0,C 180,E1 -7333.494,E2 -7333.494} C_VEL
LIN {X 0,Y 474.626,Z 762.367,A -85,B 0,C 180,E1 -7334.703,E2 -7334.703} C_VEL
LIN {X 0,Y 474.618,Z 762.367,A -85,B 0,C 180,E1 -7338.214,E2 -7338.214} C_VEL
LIN {X 0,Y 474.614,Z 762.368,A -85,B 0,C 180,E1 -7341.542,E2 -7341.542} C_VEL
LIN {X 0,Y 474.587,Z 762.528,A -85,B 0,C 180,E1 -7343.099,E2 -7343.099} C_VEL
LIN {X 0,Y 474.654,Z 763.923,A -85,B 0,C 180,E1 -7345.76,E2 -7345.76} C_VEL
LIN {X 0,Y 474.589,Z 765.197,A -85,B 0,C 180,E1 -7347.783,E2 -7347.783} C_VEL
LIN {X 0,Y 474.345,Z 767.478,A -85,B 0,C 180,E1 -7350.946,E2 -7350.946} C_VEL
LIN {X 0,Y 474.251,Z 769.562,A -85,B 0,C 180,E1 -7353.603,E2 -7353.603} C_VEL
LIN {X 0,Y 474.107,Z 772.231,A -85,B 0,C 180,E1 -7356.791,E2 -7356.791} C_VEL
LIN {X 0,Y 473.989,Z 775.132,A -85,B 0,C 180,E1 -7360.06,E2 -7360.06} C_VEL
LIN {X 0,Y 473.886,Z 777.622,A -85,B 0,C 180,E1 -7362.745,E2 -7362.745} C_VEL
LIN {X 0,Y 473.946,Z 779.891,A -85,B 0,C 180,E1 -7365,E2 -7365} C_VEL
LIN {X 0,Y 476.253,Z 790.291,A -85,B 0,C 180,E1 -7365.386,E2 -7365.386} C_VEL
LIN {X 0,Y 476.99,Z 796.614,A -85,B 0,C 180,E1 -7365.657,E2 -7365.657} C_VEL
LIN {X 0,Y 476.619,Z 808.707,A -85,B 0,C 180,E1 -7366.244,E2 -7366.244} C_VEL
LIN {X 0,Y 476.187,Z 820.326,A -85,B 0,C 180,E1 -7366.982,E2 -7366.982} C_VEL
LIN {X 0,Y 475.761,Z 831.005,A -85,B 0,C 180,E1 -7367.847,E2 -7367.847} C_VEL
LIN {X 0,Y 475.209,Z 841.61,A -85,B 0,C 180,E1 -7368.914,E2 -7368.914} C_VEL
LIN {X 0,Y 474.91,Z 850.217,A -85,B 0,C 180,E1 -7369.986,E2 -7369.986} C_VEL
LIN {X 0,Y 474.504,Z 858.562,A -85,B 0,C 180,E1 -7371.267,E2 -7371.267} C_VEL
LIN {X 0,Y 474.241,Z 864.257,A -85,B 0,C 180,E1 -7372.335,E2 -7372.335} C_VEL
LIN {X 0,Y 474.1,Z 869.794,A -85,B 0,C 180,E1 -7373.619,E2 -7373.619} C_VEL
LIN {X 0,Y 473.85,Z 874.127,A -85,B 0,C 180,E1 -7374.894,E2 -7374.894} C_VEL
LIN {X 0,Y 473.91,Z 876.405,A -85,B 0,C 180,E1 -7375.747,E2 -7375.747} C_VEL
LIN {X 0,Y 473.83,Z 878.267,A -85,B 0,C 180,E1 -7376.598,E2 -7376.598} C_VEL
LIN {X 0,Y 473.807,Z 879.673,A -85,B 0,C 180,E1 -7377.449,E2 -7377.449} C_VEL
LIN {X 0,Y 473.689,Z 881.271,A -85,B 0,C 180,E1 -7379.149,E2 -7379.149} C_VEL
LIN {X 0,Y 473.669,Z 881.495,A -85,B 0,C 180,E1 -7379.999,E2 -7379.999} C_VEL
LIN {X 0,Y 473.689,Z 881.296,A -85,B 0,C 180,E1 -7380.849,E2 -7380.849} C_VEL
LIN {X 0,Y 473.753,Z 880.694,A -85,B 0,C 180,E1 -7381.699,E2 -7381.699} C_VEL
LIN {X 0,Y 473.83,Z 878.329,A -85,B 0,C 180,E1 -7383.4,E2 -7383.4} C_VEL
LIN {X 0,Y 473.853,Z 875.432,A -85,B 0,C 180,E1 -7384.678,E2 -7384.678} C_VEL
LIN {X 0,Y 474.031,Z 871.499,A -85,B 0,C 180,E1 -7385.956,E2 -7385.956} C_VEL
LIN {X 0,Y 474.13,Z 866.434,A -85,B 0,C 180,E1 -7387.237,E2 -7387.237} C_VEL
LIN {X 0,Y 474.407,Z 860.039,A -85,B 0,C 180,E1 -7388.518,E2 -7388.518} C_VEL
LIN {X 0,Y 474.774,Z 852.052,A -85,B 0,C 180,E1 -7389.8,E2 -7389.8} C_VEL
LIN {X 0,Y 475.092,Z 843.906,A -85,B 0,C 180,E1 -7390.871,E2 -7390.871} C_VEL
LIN {X 0,Y 475.63,Z 833.966,A -85,B 0,C 180,E1 -7391.938,E2 -7391.938} C_VEL
LIN {X 0,Y 476.007,Z 822.8,A -85,B 0,C 180,E1 -7392.898,E2 -7392.898} C_VEL
LIN {X 0,Y 476.438,Z 811.775,A -85,B 0,C 180,E1 -7393.651,E2 -7393.651} C_VEL
LIN {X 0,Y 476.854,Z 799.695,A -85,B 0,C 180,E1 -7394.291,E2 -7394.291} C_VEL
LIN {X 0,Y 476.758,Z 793.439,A -85,B 0,C 180,E1 -7394.561,E2 -7394.561} C_VEL
LIN {X 0,Y 474.523,Z 781.931,A -85,B 0,C 180,E1 -7395.013,E2 -7395.013} C_VEL
LIN {X 0,Y 473.822,Z 778.535,A -85,B 0,C 180,E1 -7395.151,E2 -7395.151} C_VEL
LIN {X 0,Y 473.814,Z 775.13,A -85,B 0,C 180,E1 -7398.322,E2 -7398.322} C_VEL
LIN {X 0,Y 473.867,Z 771.523,A -85,B 0,C 180,E1 -7401.763,E2 -7401.763} C_VEL
LIN {X 0,Y 473.907,Z 768.645,A -85,B 0,C 180,E1 -7404.533,E2 -7404.533} C_VEL
LIN {X 0,Y 473.991,Z 765.745,A -85,B 0,C 180,E1 -7407.363,E2 -7407.363} C_VEL
LIN {X 0,Y 474.057,Z 762.438,A -85,B 0,C 180,E1 -7410.698,E2 -7410.698} C_VEL
LIN {X 0,Y 474.419,Z 762.392,A -85,B 0,C 180,E1 -7413.944,E2 -7413.944} C_VEL
LIN {X 0,Y 474.565,Z 762.369,A -85,B 0,C 180,E1 -7416.324,E2 -7416.324} C_VEL
LIN {X 0,Y 474.623,Z 762.364,A -85,B 0,C 180,E1 -7419.647,E2 -7419.647} C_VEL
LIN {X 0,Y 474.61,Z 762.366,A -85,B 0,C 180,E1 -7422.933,E2 -7422.933} C_VEL
LIN {X 0,Y 474.604,Z 762.365,A -85,B 0,C 180,E1 -7425.894,E2 -7425.894} C_VEL
LIN {X 0,Y 474.621,Z 762.365,A -85,B 0,C 180,E1 -7429.04,E2 -7429.04} C_VEL
LIN {X 0,Y 474.603,Z 762.366,A -85,B 0,C 180,E1 -7431.703,E2 -7431.703} C_VEL
LIN {X 0,Y 474.615,Z 762.362,A -85,B 0,C 180,E1 -7434.725,E2 -7434.725} C_VEL
LIN {X 0,Y 474.627,Z 762.363,A -85,B 0,C 180,E1 -7437.787,E2 -7437.787} C_VEL
LIN {X 0,Y 474.599,Z 762.364,A -85,B 0,C 180,E1 -7440.888,E2 -7440.888} C_VEL
LIN {X 0,Y 474.6,Z 762.365,A -85,B 0,C 180,E1 -7443.986,E2 -7443.986} C_VEL
LIN {X 0,Y 474.625,Z 762.36,A -85,B 0,C 180,E1 -7446.641,E2 -7446.641} C_VEL
LIN {X 0,Y 474.573,Z 762.368,A -85,B 0,C 180,E1 -7447.675,E2 -7447.675} C_VEL
LIN {X 0,Y 473.901,Z 762.452,A -85,B 0,C 180,E1 -7448.384,E2 -7448.384} C_VEL
LIN {X 0,Y 471.065,Z 762.809,A -85,B 0,C 180,E1 -7449.535,E2 -7449.535} C_VEL
LIN {X 0,Y 468.684,Z 763.102,A -85,B 0,C 180,E1 -7450.463,E2 -7450.463} C_VEL
LIN {X 0,Y 467.679,Z 763.227,A -85,B 0,C 180,E1 -7451.18,E2 -7451.18} C_VEL
LIN {X 0,Y 467.606,Z 763.238,A -85,B 0,C 180,E1 -7451.423,E2 -7451.423} C_VEL
LIN {X 0,Y 467.629,Z 763.233,A -85,B 0,C 180,E1 -7454.305,E2 -7454.305} C_VEL
LIN {X 0,Y 467.646,Z 763.236,A -85,B 0,C 180,E1 -7457.854,E2 -7457.854} C_VEL
LIN {X 0,Y 467.646,Z 763.23,A -85,B 0,C 180,E1 -7461.357,E2 -7461.357} C_VEL
LIN {X 0,Y 467.691,Z 763.23,A -85,B 0,C 180,E1 -7463.962,E2 -7463.962} C_VEL
LIN {X 0,Y 467.801,Z 763.21,A -85,B 0,C 180,E1 -7467.417,E2 -7467.417} C_VEL
LIN {X 0,Y 467.838,Z 763.212,A -85,B 0,C 180,E1 -7470,E2 -7470} C_VEL
LIN {X 0,Y 467.798,Z 763.211,A -85,B 0,C 180,E1 -7472.583,E2 -7472.583} C_VEL
LIN {X 0,Y 467.689,Z 763.23,A -85,B 0,C 180,E1 -7476.038,E2 -7476.038} C_VEL
LIN {X 0,Y 467.618,Z 763.234,A -85,B 0,C 180,E1 -7478.644,E2 -7478.644} C_VEL
LIN {X 0,Y 467.637,Z 763.236,A -85,B 0,C 180,E1 -7482.146,E2 -7482.146} C_VEL
LIN {X 0,Y 467.628,Z 763.232,A -85,B 0,C 180,E1 -7485.695,E2 -7485.695} C_VEL
LIN {X 0,Y 467.611,Z 763.233,A -85,B 0,C 180,E1 -7489.308,E2 -7489.308} C_VEL
LIN {X 0,Y 467.525,Z 763.247,A -85,B 0,C 180,E1 -7492.074,E2 -7492.074} C_VEL
LIN {X 0,Y 467.558,Z 763.243,A -85,B 0,C 180,E1 -7494.89,E2 -7494.89} C_VEL
LIN {X 0,Y 467.57,Z 763.24,A -85,B 0,C 180,E1 -7497.772,E2 -7497.772} C_VEL
LIN {X 0,Y 467.559,Z 763.242,A -85,B 0,C 180,E1 -7501.045,E2 -7501.045} C_VEL
LIN {X 0,Y 467.569,Z 763.242,A -85,B 0,C 180,E1 -7504.241,E2 -7504.241} C_VEL
LIN {X 0,Y 467.54,Z 763.245,A -85,B 0,C 180,E1 -7507.187,E2 -7507.187} C_VEL
LIN {X 0,Y 467.568,Z 763.242,A -85,B 0,C 180,E1 -7510.266,E2 -7510.266} C_VEL
LIN {X 0,Y 467.581,Z 763.241,A -85,B 0,C 180,E1 -7512.568,E2 -7512.568} C_VEL
LIN {X 0,Y 467.561,Z 763.245,A -85,B 0,C 180,E1 -7515.054,E2 -7515.054} C_VEL
LIN {X 0,Y 467.584,Z 763.239,A -85,B 0,C 180,E1 -7517.441,E2 -7517.441} C_VEL
LIN {X 0,Y 467.578,Z 763.243,A -85,B 0,C 180,E1 -7520.856,E2 -7520.856} C_VEL
LIN {X 0,Y 467.503,Z 763.249,A -85,B 0,C 180,E1 -7524.107,E2 -7524.107} C_VEL
LIN {X 0,Y 467.374,Z 763.268,A -85,B 0,C 180,E1 -7526.196,E2 -7526.196} C_VEL
LIN {X 0,Y 467.027,Z 763.313,A -85,B 0,C 180,E1 -7529.228,E2 -7529.228} C_VEL
LIN {X 0,Y 466.843,Z 763.567,A -85,B 0,C 180,E1 -7530.827,E2 -7530.827} C_VEL
LIN {X 0,Y 466.873,Z 766.152,A -85,B 0,C 180,E1 -7533.155,E2 -7533.155} C_VEL
LIN {X 0,Y 466.767,Z 769.266,A -85,B 0,C 180,E1 -7536.014,E2 -7536.014} C_VEL
LIN {X 0,Y 466.79,Z 772.5,A -85,B 0,C 180,E1 -7538.984,E2 -7538.984} C_VEL
LIN {X 0,Y 466.709,Z 776.329,A -85,B 0,C 180,E1 -7542.473,E2 -7542.473} C_VEL
LIN {X 0,Y 466.74,Z 778.865,A -85,B 0,C 180,E1 -7544.752,E2 -7544.752} C_VEL
LIN {X 0,Y 469.331,Z 791.137,A -85,B 0,C 180,E1 -7545.211,E2 -7545.211} C_VEL
LIN {X 0,Y 470.029,Z 797.565,A -85,B 0,C 180,E1 -7545.497,E2 -7545.497} C_VEL
LIN {X 0,Y 469.581,Z 810.278,A -85,B 0,C 180,E1 -7546.146,E2 -7546.146} C_VEL
LIN {X 0,Y 469.14,Z 821.518,A -85,B 0,C 180,E1 -7546.894,E2 -7546.894} C_VEL
LIN {X 0,Y 468.738,Z 831.968,A -85,B 0,C 180,E1 -7547.774,E2 -7547.774} C_VEL
LIN {X 0,Y 468.218,Z 841.431,A -85,B 0,C 180,E1 -7548.749,E2 -7548.749} C_VEL
LIN {X 0,Y 467.877,Z 850.087,A -85,B 0,C 180,E1 -7549.835,E2 -7549.835} C_VEL
LIN {X 0,Y 467.449,Z 858.548,A -85,B 0,C 180,E1 -7551.136,E2 -7551.136} C_VEL
LIN {X 0,Y 467.174,Z 864.291,A -85,B 0,C 180,E1 -7552.22,E2 -7552.22} C_VEL
LIN {X 0,Y 466.979,Z 870.359,A -85,B 0,C 180,E1 -7553.649,E2 -7553.649} C_VEL
LIN {X 0,Y 466.783,Z 875.509,A -85,B 0,C 180,E1 -7555.251,E2 -7555.251} C_VEL
LIN {X 0,Y 466.762,Z 878.486,A -85,B 0,C 180,E1 -7556.548,E2 -7556.548} C_VEL
LIN {X 0,Y 466.681,Z 879.941,A -85,B 0,C 180,E1 -7557.411,E2 -7557.411} C_VEL
LIN {X 0,Y 466.688,Z 880.961,A -85,B 0,C 180,E1 -7558.275,E2 -7558.275} C_VEL
LIN {X 0,Y 466.599,Z 881.859,A -85,B 0,C 180,E1 -7560.001,E2 -7560.001} C_VEL
LIN {X 0,Y 466.62,Z 881.683,A -85,B 0,C 180,E1 -7560.864,E2 -7560.864} C_VEL
LIN {X 0,Y 466.689,Z 881.108,A -85,B 0,C 180,E1 -7561.727,E2 -7561.727} C_VEL
LIN {X 0,Y 466.708,Z 880.154,A -85,B 0,C 180,E1 -7562.59,E2 -7562.59} C_VEL
LIN {X 0,Y 466.765,Z 878.793,A -85,B 0,C 180,E1 -7563.454,E2 -7563.454} C_VEL
LIN {X 0,Y 466.812,Z 875.93,A -85,B 0,C 180,E1 -7564.751,E2 -7564.751} C_VEL
LIN {X 0,Y 467.044,Z 870.75,A -85,B 0,C 180,E1 -7566.398,E2 -7566.398} C_VEL
LIN {X 0,Y 467.185,Z 864.985,A -85,B 0,C 180,E1 -7567.782,E2 -7567.782} C_VEL
LIN {X 0,Y 467.516,Z 858.091,A -85,B 0,C 180,E1 -7569.083,E2 -7569.083} C_VEL
LIN {X 0,Y 467.945,Z 849.489,A -85,B 0,C 180,E1 -7570.384,E2 -7570.384} C_VEL
LIN {X 0,Y 468.393,Z 840.666,A -85,B 0,C 180,E1 -7571.468,E2 -7571.468} C_VEL
LIN {X 0,Y 468.884,Z 829.981,A -85,B 0,C 180,E1 -7572.526,E2 -7572.526} C_VEL
LIN {X 0,Y 469.28,Z 818.69,A -85,B 0,C 180,E1 -7573.423,E2 -7573.423} C_VEL
LIN {X 0,Y 469.797,Z 806.313,A -85,B 0,C 180,E1 -7574.181,E2 -7574.181} C_VEL
LIN {X 0,Y 470.04,Z 795.978,A -85,B 0,C 180,E1 -7574.671,E2 -7574.671} C_VEL
LIN {X 0,Y 468.236,Z 785.699,A -85,B 0,C 180,E1 -7575.107,E2 -7575.107} C_VEL
LIN {X 0,Y 466.819,Z 779.915,A -85,B 0,C 180,E1 -7575.33,E2 -7575.33} C_VEL
LIN {X 0,Y 466.83,Z 776.498,A -85,B 0,C 180,E1 -7578.477,E2 -7578.477} C_VEL
LIN {X 0,Y 466.821,Z 773.486,A -85,B 0,C 180,E1 -7581.182,E2 -7581.182} C_VEL
LIN {X 0,Y 466.861,Z 770.392,A -85,B 0,C 180,E1 -7583.983,E2 -7583.983} C_VEL
LIN {X 0,Y 466.892,Z 766.953,A -85,B 0,C 180,E1 -7586.846,E2 -7586.846} C_VEL
LIN {X 0,Y 466.864,Z 763.335,A -85,B 0,C 180,E1 -7589.787,E2 -7589.787} C_VEL
LIN {X 0,Y 467.251,Z 763.286,A -85,B 0,C 180,E1 -7592.785,E2 -7592.785} C_VEL
LIN {X 0,Y 467.505,Z 763.251,A -85,B 0,C 180,E1 -7595.729,E2 -7595.729} C_VEL
LIN {X 0,Y 467.563,Z 763.243,A -85,B 0,C 180,E1 -7598.591,E2 -7598.591} C_VEL
LIN {X 0,Y 467.577,Z 763.243,A -85,B 0,C 180,E1 -7601.404,E2 -7601.404} C_VEL
LIN {X 0,Y 467.575,Z 763.245,A -85,B 0,C 180,E1 -7605.053,E2 -7605.053} C_VEL
LIN {X 0,Y 467.594,Z 763.24,A -85,B 0,C 180,E1 -7607.44,E2 -7607.44} C_VEL
LIN {X 0,Y 467.606,Z 763.448,A -85,B 0,C 180,E1 -7609.314,E2 -7609.314} C_VEL
LIN {X 0,Y 468.734,Z 769.592,A -85,B 0,C 180,E1 -7612.067,E2 -7612.067} C_VEL
LIN {X 0,Y 469.384,Z 774.777,A -85,B 0,C 180,E1 -7614.272,E2 -7614.272} C_VEL
LIN {X 0,Y 469.039,Z 781.753,A -85,B 0,C 180,E1 -7617.045,E2 -7617.045} C_VEL
LIN {X 0,Y 468.609,Z 789.015,A -85,B 0,C 180,E1 -7619.84,E2 -7619.84} C_VEL
LIN {X 0,Y 468.23,Z 796.87,A -85,B 0,C 180,E1 -7622.769,E2 -7622.769} C_VEL
LIN {X 0,Y 467.93,Z 804.686,A -85,B 0,C 180,E1 -7625.604,E2 -7625.604} C_VEL
LIN {X 0,Y 467.567,Z 813.895,A -85,B 0,C 180,E1 -7628.854,E2 -7628.854} C_VEL
LIN {X 0,Y 467.287,Z 823.138,A -85,B 0,C 180,E1 -7632.042,E2 -7632.042} C_VEL
LIN {X 0,Y 467.117,Z 830.714,A -85,B 0,C 180,E1 -7634.611,E2 -7634.611} C_VEL
LIN {X 0,Y 469.205,Z 844.659,A -85,B 0,C 180,E1 -7635.059,E2 -7635.059} C_VEL
LIN {X 0,Y 469.972,Z 851.134,A -85,B 0,C 180,E1 -7635.328,E2 -7635.328} C_VEL
LIN {X 0,Y 469.546,Z 863.568,A -85,B 0,C 180,E1 -7635.923,E2 -7635.923} C_VEL
LIN {X 0,Y 469.02,Z 875.572,A -85,B 0,C 180,E1 -7636.68,E2 -7636.68} C_VEL
LIN {X 0,Y 468.522,Z 886.877,A -85,B 0,C 180,E1 -7637.594,E2 -7637.594} C_VEL
LIN {X 0,Y 468.124,Z 896.227,A -85,B 0,C 180,E1 -7638.526,E2 -7638.526} C_VEL
LIN {X 0,Y 467.661,Z 905.197,A -85,B 0,C 180,E1 -7639.611,E2 -7639.611} C_VEL
LIN {X 0,Y 467.288,Z 913.976,A -85,B 0,C 180,E1 -7640.914,E2 -7640.914} C_VEL
LIN {X 0,Y 467.008,Z 920.981,A -85,B 0,C 180,E1 -7642.216,E2 -7642.216} C_VEL
LIN {X 0,Y 466.823,Z 926.65,A -85,B 0,C 180,E1 -7643.532,E2 -7643.532} C_VEL
LIN {X 0,Y 466.779,Z 931.001,A -85,B 0,C 180,E1 -7644.817,E2 -7644.817} C_VEL
LIN {X 0,Y 466.665,Z 933.323,A -85,B 0,C 180,E1 -7645.682,E2 -7645.682} C_VEL
LIN {X 0,Y 466.727,Z 935.216,A -85,B 0,C 180,E1 -7646.547,E2 -7646.547} C_VEL
LIN {X 0,Y 466.684,Z 937.636,A -85,B 0,C 180,E1 -7648.274,E2 -7648.274} C_VEL
LIN {X 0,Y 466.62,Z 938.238,A -85,B 0,C 180,E1 -7649.137,E2 -7649.137} C_VEL
LIN {X 0,Y 466.599,Z 938.444,A -85,B 0,C 180,E1 -7650,E2 -7650} C_VEL
LIN {X 0,Y 466.62,Z 938.213,A -85,B 0,C 180,E1 -7650.863,E2 -7650.863} C_VEL
LIN {X 0,Y 466.684,Z 937.587,A -85,B 0,C 180,E1 -7651.726,E2 -7651.726} C_VEL
LIN {X 0,Y 466.746,Z 935.105,A -85,B 0,C 180,E1 -7653.453,E2 -7653.453} C_VEL
LIN {X 0,Y 466.704,Z 932.073,A -85,B 0,C 180,E1 -7654.751,E2 -7654.751} C_VEL
LIN {X 0,Y 466.811,Z 927.982,A -85,B 0,C 180,E1 -7656.05,E2 -7656.05} C_VEL
LIN {X 0,Y 466.959,Z 921.692,A -85,B 0,C 180,E1 -7657.567,E2 -7657.567} C_VEL
LIN {X 0,Y 467.229,Z 914.818,A -85,B 0,C 180,E1 -7658.869,E2 -7658.869} C_VEL
LIN {X 0,Y 467.559,Z 906.29,A -85,B 0,C 180,E1 -7660.173,E2 -7660.173} C_VEL
LIN {X 0,Y 467.993,Z 897.527,A -85,B 0,C 180,E1 -7661.258,E2 -7661.258} C_VEL
LIN {X 0,Y 468.482,Z 887.177,A -85,B 0,C 180,E1 -7662.304,E2 -7662.304} C_VEL
LIN {X 0,Y 468.893,Z 876.095,A -85,B 0,C 180,E1 -7663.213,E2 -7663.213} C_VEL
LIN {X 0,Y 469.384,Z 864.353,A -85,B 0,C 180,E1 -7663.971,E2 -7663.971} C_VEL
LIN {X 0,Y 469.903,Z 851.082,A -85,B 0,C 180,E1 -7664.619,E2 -7664.619} C_VEL
LIN {X 0,Y 468.158,Z 838.029,A -85,B 0,C 180,E1 -7665.134,E2 -7665.134} C_VEL
LIN {X 0,Y 467.097,Z 829.576,A -85,B 0,C 180,E1 -7665.384,E2 -7665.384} C_VEL
LIN {X 0,Y 467.278,Z 818.754,A -85,B 0,C 180,E1 -7668.93,E2 -7668.93} C_VEL
LIN {X 0,Y 467.496,Z 809.395,A -85,B 0,C 180,E1 -7672.076,E2 -7672.076} C_VEL
LIN {X 0,Y 467.793,Z 800.273,A -85,B 0,C 180,E1 -7675.266,E2 -7675.266} C_VEL
LIN {X 0,Y 468.094,Z 792.193,A -85,B 0,C 180,E1 -7678.226,E2 -7678.226} C_VEL
LIN {X 0,Y 468.631,Z 783.539,A -85,B 0,C 180,E1 -7681.661,E2 -7681.661} C_VEL
LIN {X 0,Y 469.122,Z 777.125,A -85,B 0,C 180,E1 -7684.515,E2 -7684.515} C_VEL
LIN {X 0,Y 469.296,Z 774.094,A -85,B 0,C 180,E1 -7686.032,E2 -7686.032} C_VEL
LIN {X 0,Y 468.887,Z 770.868,A -85,B 0,C 180,E1 -7687.918,E2 -7687.918} C_VEL
LIN {X 0,Y 468.392,Z 767.694,A -85,B 0,C 180,E1 -7690.181,E2 -7690.181} C_VEL
LIN {X 0,Y 467.919,Z 765.173,A -85,B 0,C 180,E1 -7692.61,E2 -7692.61} C_VEL
LIN {X 0,Y 467.623,Z 763.572,A -85,B 0,C 180,E1 -7695.059,E2 -7695.059} C_VEL
LIN {X 0,Y 467.564,Z 763.246,A -85,B 0,C 180,E1 -7697.436,E2 -7697.436} C_VEL
LIN {X 0,Y 467.574,Z 763.245,A -85,B 0,C 180,E1 -7700.047,E2 -7700.047} C_VEL
LIN {X 0,Y 467.567,Z 763.388,A -85,B 0,C 180,E1 -7701.955,E2 -7701.955} C_VEL
LIN {X 0,Y 467.66,Z 764.309,A -85,B 0,C 180,E1 -7704.244,E2 -7704.244} C_VEL
LIN {X 0,Y 467.611,Z 766.003,A -85,B 0,C 180,E1 -7707.316,E2 -7707.316} C_VEL
LIN {X 0,Y 467.372,Z 767.992,A -85,B 0,C 180,E1 -7710.248,E2 -7710.248} C_VEL
LIN {X 0,Y 467.212,Z 770.185,A -85,B 0,C 180,E1 -7713.174,E2 -7713.174} C_VEL
LIN {X 0,Y 467.087,Z 772.975,A -85,B 0,C 180,E1 -7716.612,E2 -7716.612} C_VEL
LIN {X 0,Y 466.946,Z 775.694,A -85,B 0,C 180,E1 -7719.746,E2 -7719.746} C_VEL
LIN {X 0,Y 466.836,Z 778.181,A -85,B 0,C 180,E1 -7722.476,E2 -7722.476} C_VEL
LIN {X 0,Y 466.901,Z 780.447,A -85,B 0,C 180,E1 -7724.77,E2 -7724.77} C_VEL
LIN {X 0,Y 469.445,Z 791.663,A -85,B 0,C 180,E1 -7725.21,E2 -7725.21} C_VEL
LIN {X 0,Y 470.13,Z 796.868,A -85,B 0,C 180,E1 -7725.443,E2 -7725.443} C_VEL
LIN {X 0,Y 469.741,Z 808.948,A -85,B 0,C 180,E1 -7726.039,E2 -7726.039} C_VEL
LIN {X 0,Y 469.282,Z 820.321,A -85,B 0,C 180,E1 -7726.768,E2 -7726.768} C_VEL
LIN {X 0,Y 468.843,Z 831.316,A -85,B 0,C 180,E1 -7727.665,E2 -7727.665} C_VEL
LIN {X 0,Y 468.247,Z 841.944,A -85,B 0,C 180,E1 -7728.748,E2 -7728.748} C_VEL
LIN {X 0,Y 467.915,Z 850.575,A -85,B 0,C 180,E1 -7729.834,E2 -7729.834} C_VEL
LIN {X 0,Y 467.482,Z 858.951,A -85,B 0,C 180,E1 -7731.135,E2 -7731.135} C_VEL
LIN {X 0,Y 467.208,Z 864.662,A -85,B 0,C 180,E1 -7732.218,E2 -7732.218} C_VEL
LIN {X 0,Y 467.055,Z 870.462,A -85,B 0,C 180,E1 -7733.59,E2 -7733.59} C_VEL
LIN {X 0,Y 466.793,Z 874.555,A -85,B 0,C 180,E1 -7734.816,E2 -7734.816} C_VEL
LIN {X 0,Y 466.841,Z 876.837,A -85,B 0,C 180,E1 -7735.682,E2 -7735.682} C_VEL
LIN {X 0,Y 466.766,Z 878.7,A -85,B 0,C 180,E1 -7736.546,E2 -7736.546} C_VEL
LIN {X 0,Y 466.737,Z 880.109,A -85,B 0,C 180,E1 -7737.41,E2 -7737.41} C_VEL
LIN {X 0,Y 466.69,Z 881.098,A -85,B 0,C 180,E1 -7738.273,E2 -7738.273} C_VEL
LIN {X 0,Y 466.598,Z 881.925,A -85,B 0,C 180,E1 -7739.999,E2 -7739.999} C_VEL
LIN {X 0,Y 466.62,Z 881.721,A -85,B 0,C 180,E1 -7740.862,E2 -7740.862} C_VEL
LIN {X 0,Y 466.689,Z 881.11,A -85,B 0,C 180,E1 -7741.725,E2 -7741.725} C_VEL
LIN {X 0,Y 466.764,Z 878.732,A -85,B 0,C 180,E1 -7743.452,E2 -7743.452} C_VEL
LIN {X 0,Y 466.774,Z 875.82,A -85,B 0,C 180,E1 -7744.749,E2 -7744.749} C_VEL
LIN {X 0,Y 466.985,Z 871.868,A -85,B 0,C 180,E1 -7746.046,E2 -7746.046} C_VEL
LIN {X 0,Y 467.111,Z 865.787,A -85,B 0,C 180,E1 -7747.564,E2 -7747.564} C_VEL
LIN {X 0,Y 467.442,Z 859.125,A -85,B 0,C 180,E1 -7748.864,E2 -7748.864} C_VEL
LIN {X 0,Y 467.833,Z 850.857,A -85,B 0,C 180,E1 -7750.166,E2 -7750.166} C_VEL
LIN {X 0,Y 468.202,Z 842.365,A -85,B 0,C 180,E1 -7751.252,E2 -7751.252} C_VEL
LIN {X 0,Y 468.774,Z 831.935,A -85,B 0,C 180,E1 -7752.329,E2 -7752.329} C_VEL
LIN {X 0,Y 469.183,Z 820.5,A -85,B 0,C 180,E1 -7753.283,E2 -7753.283} C_VEL
LIN {X 0,Y 469.677,Z 808.252,A -85,B 0,C 180,E1 -7754.072,E2 -7754.072} C_VEL
LIN {X 0,Y 470.048,Z 796.052,A -85,B 0,C 180,E1 -7754.669,E2 -7754.669} C_VEL
LIN {X 0,Y 468.357,Z 785.954,A -85,B 0,C 180,E1 -7755.097,E2 -7755.097} C_VEL
LIN {X 0,Y 466.734,Z 778.901,A -85,B 0,C 180,E1 -7755.36,E2 -7755.36} C_VEL
LIN {X 0,Y 466.739,Z 775.607,A -85,B 0,C 180,E1 -7758.443,E2 -7758.443} C_VEL
LIN {X 0,Y 466.787,Z 772.738,A -85,B 0,C 180,E1 -7761.182,E2 -7761.182} C_VEL
LIN {X 0,Y 466.852,Z 769.841,A -85,B 0,C 180,E1 -7763.981,E2 -7763.981} C_VEL
LIN {X 0,Y 466.915,Z 766.916,A -85,B 0,C 180,E1 -7766.843,E2 -7766.843} C_VEL
LIN {X 0,Y 466.927,Z 763.942,A -85,B 0,C 180,E1 -7769.781,E2 -7769.781} C_VEL
LIN {X 0,Y 467.028,Z 763.313,A -85,B 0,C 180,E1 -7770.934,E2 -7770.934} C_VEL
LIN {X 0,Y 467.407,Z 763.266,A -85,B 0,C 180,E1 -7774.209,E2 -7774.209} C_VEL
LIN {X 0,Y 467.536,Z 763.248,A -85,B 0,C 180,E1 -7777.184,E2 -7777.184} C_VEL
LIN {X 0,Y 467.573,Z 763.24,A -85,B 0,C 180,E1 -7780.264,E2 -7780.264} C_VEL
LIN {X 0,Y 467.582,Z 763.239,A -85,B 0,C 180,E1 -7782.566,E2 -7782.566} C_VEL
LIN {X 0,Y 467.565,Z 763.245,A -85,B 0,C 180,E1 -7785.052,E2 -7785.052} C_VEL
LIN {X 0,Y 467.583,Z 763.242,A -85,B 0,C 180,E1 -7787.439,E2 -7787.439} C_VEL
LIN {X 0,Y 467.569,Z 763.241,A -85,B 0,C 180,E1 -7790.854,E2 -7790.854} C_VEL
LIN {X 0,Y 467.552,Z 763.242,A -85,B 0,C 180,E1 -7794.26,E2 -7794.26} C_VEL
LIN {X 0,Y 467.572,Z 763.245,A -85,B 0,C 180,E1 -7797.321,E2 -7797.321} C_VEL
LIN {X 0,Y 467.549,Z 763.242,A -85,B 0,C 180,E1 -7800.67,E2 -7800.67} C_VEL
LIN {X 0,Y 467.555,Z 763.244,A -85,B 0,C 180,E1 -7803.196,E2 -7803.196} C_VEL
LIN {X 0,Y 467.58,Z 763.238,A -85,B 0,C 180,E1 -7806.469,E2 -7806.469} C_VEL
LIN {X 0,Y 467.612,Z 763.239,A -85,B 0,C 180,E1 -7809.777,E2 -7809.777} C_VEL
LIN {X 0,Y 467.606,Z 763.238,A -85,B 0,C 180,E1 -7811.423,E2 -7811.423} C_VEL
LIN {X 0,Y 466.962,Z 763.324,A -85,B 0,C 180,E1 -7812.142,E2 -7812.142} C_VEL
LIN {X 0,Y 464.114,Z 763.677,A -85,B 0,C 180,E1 -7813.31,E2 -7813.31} C_VEL
LIN {X 0,Y 461.684,Z 763.974,A -85,B 0,C 180,E1 -7814.252,E2 -7814.252} C_VEL
LIN {X 0,Y 460.629,Z 764.103,A -85,B 0,C 180,E1 -7814.979,E2 -7814.979} C_VEL
LIN {X 0,Y 460.539,Z 764.115,A -85,B 0,C 180,E1 -7815.226,E2 -7815.226} C_VEL
LIN {X 0,Y 460.598,Z 764.108,A -85,B 0,C 180,E1 -7818.559,E2 -7818.559} C_VEL
LIN {X 0,Y 460.598,Z 764.107,A -85,B 0,C 180,E1 -7821.223,E2 -7821.223} C_VEL
LIN {X 0,Y 460.657,Z 764.107,A -85,B 0,C 180,E1 -7823.869,E2 -7823.869} C_VEL
LIN {X 0,Y 460.744,Z 764.089,A -85,B 0,C 180,E1 -7827.377,E2 -7827.377} C_VEL
LIN {X 0,Y 460.807,Z 764.088,A -85,B 0,C 180,E1 -7830,E2 -7830} C_VEL
LIN {X 0,Y 460.742,Z 764.09,A -85,B 0,C 180,E1 -7832.623,E2 -7832.623} C_VEL
LIN {X 0,Y 460.655,Z 764.107,A -85,B 0,C 180,E1 -7836.131,E2 -7836.131} C_VEL
LIN {X 0,Y 460.574,Z 764.111,A -85,B 0,C 180,E1 -7838.777,E2 -7838.777} C_VEL
LIN {X 0,Y 460.587,Z 764.114,A -85,B 0,C 180,E1 -7842.435,E2 -7842.435} C_VEL
LIN {X 0,Y 460.591,Z 764.111,A -85,B 0,C 180,E1 -7845.998,E2 -7845.998} C_VEL
LIN {X 0,Y 460.557,Z 764.113,A -85,B 0,C 180,E1 -7849.616,E2 -7849.616} C_VEL
LIN {X 0,Y 460.501,Z 764.126,A -85,B 0,C 180,E1 -7852.429,E2 -7852.429} C_VEL
LIN {X 0,Y 460.526,Z 764.117,A -85,B 0,C 180,E1 -7855.794,E2 -7855.794} C_VEL
LIN {X 0,Y 460.517,Z 764.12,A -85,B 0,C 180,E1 -7858.235,E2 -7858.235} C_VEL
LIN {X 0,Y 460.512,Z 764.119,A -85,B 0,C 180,E1 -7861.283,E2 -7861.283} C_VEL
LIN {X 0,Y 460.516,Z 764.122,A -85,B 0,C 180,E1 -7864.505,E2 -7864.505} C_VEL
LIN {X 0,Y 460.494,Z 764.121,A -85,B 0,C 180,E1 -7867.624,E2 -7867.624} C_VEL
LIN {X 0,Y 460.532,Z 764.118,A -85,B 0,C 180,E1 -7870.27,E2 -7870.27} C_VEL
LIN {X 0,Y 460.493,Z 764.122,A -85,B 0,C 180,E1 -7873.376,E2 -7873.376} C_VEL
LIN {X 0,Y 460.494,Z 764.124,A -85,B 0,C 180,E1 -7876.626,E2 -7876.626} C_VEL
LIN {X 0,Y 460.537,Z 764.116,A -85,B 0,C 180,E1 -7879.732,E2 -7879.732} C_VEL
LIN {X 0,Y 460.494,Z 764.123,A -85,B 0,C 180,E1 -7882.525,E2 -7882.525} C_VEL
LIN {X 0,Y 460.387,Z 764.141,A -85,B 0,C 180,E1 -7885.612,E2 -7885.612} C_VEL
LIN {X 0,Y 460.181,Z 764.166,A -85,B 0,C 180,E1 -7887.689,E2 -7887.689} C_VEL
LIN {X 0,Y 459.776,Z 764.217,A -85,B 0,C 180,E1 -7890.717,E2 -7890.717} C_VEL
LIN {X 0,Y 459.794,Z 767.306,A -85,B 0,C 180,E1 -7893.689,E2 -7893.689} C_VEL
LIN {X 0,Y 459.73,Z 770.475,A -85,B 0,C 180,E1 -7896.581,E2 -7896.581} C_VEL
LIN {X 0,Y 459.705,Z 773.564,A -85,B 0,C 180,E1 -7899.414,E2 -7899.414} C_VEL
LIN {X 0,Y 459.641,Z 776.592,A -85,B 0,C 180,E1 -7902.195,E2 -7902.195} C_VEL
LIN {X 0,Y 459.649,Z 779.133,A -85,B 0,C 180,E1 -7904.513,E2 -7904.513} C_VEL
LIN {X 0,Y 462.494,Z 792.334,A -85,B 0,C 180,E1 -7905.03,E2 -7905.03} C_VEL
LIN {X 0,Y 463.165,Z 797.689,A -85,B 0,C 180,E1 -7905.277,E2 -7905.277} C_VEL
LIN {X 0,Y 462.688,Z 810.425,A -85,B 0,C 180,E1 -7905.935,E2 -7905.935} C_VEL
LIN {X 0,Y 462.217,Z 821.578,A -85,B 0,C 180,E1 -7906.686,E2 -7906.686} C_VEL
LIN {X 0,Y 461.8,Z 832.246,A -85,B 0,C 180,E1 -7907.594,E2 -7907.594} C_VEL
LIN {X 0,Y 461.269,Z 841.674,A -85,B 0,C 180,E1 -7908.577,E2 -7908.577} C_VEL
LIN {X 0,Y 460.882,Z 850.357,A -85,B 0,C 180,E1 -7909.679,E2 -7909.679} C_VEL
LIN {X 0,Y 460.444,Z 858.851,A -85,B 0,C 180,E1 -7911,E2 -7911} C_VEL
LIN {X 0,Y 460.104,Z 865.619,A -85,B 0,C 180,E1 -7912.32,E2 -7912.32} C_VEL
LIN {X 0,Y 459.934,Z 871.827,A -85,B 0,C 180,E1 -7913.861,E2 -7913.861} C_VEL
LIN {X 0,Y 459.704,Z 875.882,A -85,B 0,C 180,E1 -7915.178,E2 -7915.178} C_VEL
LIN {X 0,Y 459.698,Z 878.874,A -85,B 0,C 180,E1 -7916.495,E2 -7916.495} C_VEL
LIN {X 0,Y 459.605,Z 880.34,A -85,B 0,C 180,E1 -7917.372,E2 -7917.372} C_VEL
LIN {X 0,Y 459.624,Z 881.365,A -85,B 0,C 180,E1 -7918.248,E2 -7918.248} C_VEL
LIN {X 0,Y 459.53,Z 882.275,A -85,B 0,C 180,E1 -7920.001,E2 -7920.001} C_VEL
LIN {X 0,Y 459.553,Z 882.1,A -85,B 0,C 180,E1 -7920.877,E2 -7920.877} C_VEL
LIN {X 0,Y 459.627,Z 881.526,A -85,B 0,C 180,E1 -7921.753,E2 -7921.753} C_VEL
LIN {X 0,Y 459.629,Z 880.574,A -85,B 0,C 180,E1 -7922.63,E2 -7922.63} C_VEL
LIN {X 0,Y 459.702,Z 879.208,A -85,B 0,C 180,E1 -7923.507,E2 -7923.507} C_VEL
LIN {X 0,Y 459.75,Z 876.338,A -85,B 0,C 180,E1 -7924.824,E2 -7924.824} C_VEL
LIN {X 0,Y 460,Z 871.384,A -85,B 0,C 180,E1 -7926.429,E2 -7926.429} C_VEL
LIN {X 0,Y 460.173,Z 865.362,A -85,B 0,C 180,E1 -7927.901,E2 -7927.901} C_VEL
LIN {X 0,Y 460.505,Z 858.441,A -85,B 0,C 180,E1 -7929.222,E2 -7929.222} C_VEL
LIN {X 0,Y 460.974,Z 849.821,A -85,B 0,C 180,E1 -7930.543,E2 -7930.543} C_VEL
LIN {X 0,Y 461.447,Z 840.987,A -85,B 0,C 180,E1 -7931.643,E2 -7931.643} C_VEL
LIN {X 0,Y 461.955,Z 830.544,A -85,B 0,C 180,E1 -7932.694,E2 -7932.694} C_VEL
LIN {X 0,Y 462.319,Z 820.636,A -85,B 0,C 180,E1 -7933.506,E2 -7933.506} C_VEL
LIN {X 0,Y 462.832,Z 808.651,A -85,B 0,C 180,E1 -7934.286,E2 -7934.286} C_VEL
LIN {X 0,Y 463.219,Z 797.603,A -85,B 0,C 180,E1 -7934.835,E2 -7934.835} C_VEL
LIN {X 0,Y 461.704,Z 788.223,A -85,B 0,C 180,E1 -7935.255,E2 -7935.255} C_VEL
LIN {X 0,Y 459.743,Z 780.421,A -85,B 0,C 180,E1 -7935.564,E2 -7935.564} C_VEL
LIN {X 0,Y 459.77,Z 776.988,A -85,B 0,C 180,E1 -7938.724,E2 -7938.724} C_VEL
LIN {X 0,Y 459.755,Z 773.896,A -85,B 0,C 180,E1 -7941.524,E2 -7941.524} C_VEL
LIN {X 0,Y 459.803,Z 770.675,A -85,B 0,C 180,E1 -7944.375,E2 -7944.375} C_VEL
LIN {X 0,Y 459.822,Z 768.323,A -85,B 0,C 180,E1 -7946.312,E2 -7946.312} C_VEL
LIN {X 0,Y 459.801,Z 764.512,A -85,B 0,C 180,E1 -7949.397,E2 -7949.397} C_VEL
LIN {X 0,Y 460.023,Z 764.186,A -85,B 0,C 180,E1 -7951.295,E2 -7951.295} C_VEL
LIN {X 0,Y 460.384,Z 764.141,A -85,B 0,C 180,E1 -7954.391,E2 -7954.391} C_VEL
LIN {X 0,Y 460.502,Z 764.123,A -85,B 0,C 180,E1 -7957.624,E2 -7957.624} C_VEL
LIN {X 0,Y 460.539,Z 764.117,A -85,B 0,C 180,E1 -7960.269,E2 -7960.269} C_VEL
LIN {X 0,Y 460.514,Z 764.122,A -85,B 0,C 180,E1 -7963.374,E2 -7963.374} C_VEL
LIN {X 0,Y 460.505,Z 764.123,A -85,B 0,C 180,E1 -7966.625,E2 -7966.625} C_VEL
LIN {X 0,Y 460.569,Z 764.24,A -85,B 0,C 180,E1 -7968.993,E2 -7968.993} C_VEL
LIN {X 0,Y 461.963,Z 772.016,A -85,B 0,C 180,E1 -7972.516,E2 -7972.516} C_VEL
LIN {X 0,Y 462.408,Z 775.939,A -85,B 0,C 180,E1 -7974.206,E2 -7974.206} C_VEL
LIN {X 0,Y 461.995,Z 783.648,A -85,B 0,C 180,E1 -7977.314,E2 -7977.314} C_VEL
LIN {X 0,Y 461.55,Z 791.123,A -85,B 0,C 180,E1 -7980.221,E2 -7980.221} C_VEL
LIN {X 0,Y 461.147,Z 799.236,A -85,B 0,C 180,E1 -7983.283,E2 -7983.283} C_VEL
LIN {X 0,Y 460.776,Z 807.264,A -85,B 0,C 180,E1 -7986.229,E2 -7986.229} C_VEL
LIN {X 0,Y 460.435,Z 816.263,A -85,B 0,C 180,E1 -7989.447,E2 -7989.447} C_VEL
LIN {X 0,Y 460.148,Z 825.477,A -85,B 0,C 180,E1 -7992.673,E2 -7992.673} C_VEL
LIN {X 0,Y 460.046,Z 830.551,A -85,B 0,C 180,E1 -7994.384,E2 -7994.384} C_VEL
LIN {X 0,Y 462.127,Z 844.344,A -85,B 0,C 180,E1 -7994.835,E2 -7994.835} C_VEL
LIN {X 0,Y 463.039,Z 851.853,A -85,B 0,C 180,E1 -7995.159,E2 -7995.159} C_VEL
LIN {X 0,Y 462.522,Z 864.944,A -85,B 0,C 180,E1 -7995.817,E2 -7995.817} C_VEL
LIN {X 0,Y 461.994,Z 876.519,A -85,B 0,C 180,E1 -7996.586,E2 -7996.586} C_VEL
LIN {X 0,Y 461.483,Z 887.629,A -85,B 0,C 180,E1 -7997.522,E2 -7997.522} C_VEL
LIN {X 0,Y 461.012,Z 897.68,A -85,B 0,C 180,E1 -7998.569,E2 -7998.569} C_VEL
LIN {X 0,Y 460.555,Z 906.341,A -85,B 0,C 180,E1 -7999.671,E2 -7999.671} C_VEL
LIN {X 0,Y 460.168,Z 914.762,A -85,B 0,C 180,E1 -8000.994,E2 -8000.994} C_VEL
LIN {X 0,Y 459.898,Z 921.549,A -85,B 0,C 180,E1 -8002.316,E2 -8002.316} C_VEL
LIN {X 0,Y 459.719,Z 927.777,A -85,B 0,C 180,E1 -8003.857,E2 -8003.857} C_VEL
LIN {X 0,Y 459.634,Z 931.813,A -85,B 0,C 180,E1 -8005.176,E2 -8005.176} C_VEL
LIN {X 0,Y 459.625,Z 934.79,A -85,B 0,C 180,E1 -8006.493,E2 -8006.493} C_VEL
LIN {X 0,Y 459.573,Z 936.207,A -85,B 0,C 180,E1 -8007.37,E2 -8007.37} C_VEL
LIN {X 0,Y 459.62,Z 937.214,A -85,B 0,C 180,E1 -8008.248,E2 -8008.248} C_VEL
LIN {X 0,Y 459.554,Z 937.814,A -85,B 0,C 180,E1 -8009.124,E2 -8009.124} C_VEL
LIN {X 0,Y 459.53,Z 938.018,A -85,B 0,C 180,E1 -8010,E2 -8010} C_VEL
LIN {X 0,Y 459.554,Z 937.783,A -85,B 0,C 180,E1 -8010.876,E2 -8010.876} C_VEL
LIN {X 0,Y 459.62,Z 937.148,A -85,B 0,C 180,E1 -8011.752,E2 -8011.752} C_VEL
LIN {X 0,Y 459.573,Z 936.1,A -85,B 0,C 180,E1 -8012.63,E2 -8012.63} C_VEL
LIN {X 0,Y 459.657,Z 934.647,A -85,B 0,C 180,E1 -8013.506,E2 -8013.506} C_VEL
LIN {X 0,Y 459.635,Z 931.599,A -85,B 0,C 180,E1 -8014.824,E2 -8014.824} C_VEL
LIN {X 0,Y 459.727,Z 927.484,A -85,B 0,C 180,E1 -8016.143,E2 -8016.143} C_VEL
LIN {X 0,Y 459.898,Z 921.156,A -85,B 0,C 180,E1 -8017.684,E2 -8017.684} C_VEL
LIN {X 0,Y 460.165,Z 914.25,A -85,B 0,C 180,E1 -8019.007,E2 -8019.007} C_VEL
LIN {X 0,Y 460.525,Z 905.685,A -85,B 0,C 180,E1 -8020.33,E2 -8020.33} C_VEL
LIN {X 0,Y 460.996,Z 896.881,A -85,B 0,C 180,E1 -8021.431,E2 -8021.431} C_VEL
LIN {X 0,Y 461.484,Z 886.75,A -85,B 0,C 180,E1 -8022.469,E2 -8022.469} C_VEL
LIN {X 0,Y 461.949,Z 875.376,A -85,B 0,C 180,E1 -8023.416,E2 -8023.416} C_VEL
LIN {X 0,Y 462.446,Z 863.609,A -85,B 0,C 180,E1 -8024.185,E2 -8024.185} C_VEL
LIN {X 0,Y 462.916,Z 850.349,A -85,B 0,C 180,E1 -8024.845,E2 -8024.845} C_VEL
LIN {X 0,Y 461.047,Z 837.188,A -85,B 0,C 180,E1 -8025.379,E2 -8025.379} C_VEL
LIN {X 0,Y 460.018,Z 829.047,A -85,B 0,C 180,E1 -8025.628,E2 -8025.628} C_VEL
LIN {X 0,Y 460.196,Z 819.671,A -85,B 0,C 180,E1 -8028.763,E2 -8028.763} C_VEL
LIN {X 0,Y 460.413,Z 810.333,A -85,B 0,C 180,E1 -8031.961,E2 -8031.961} C_VEL
LIN {X 0,Y 460.676,Z 802.344,A -85,B 0,C 180,E1 -8034.805,E2 -8034.805} C_VEL
LIN {X 0,Y 461.025,Z 794.16,A -85,B 0,C 180,E1 -8037.849,E2 -8037.849} C_VEL
LIN {X 0,Y 461.517,Z 785.86,A -85,B 0,C 180,E1 -8041.182,E2 -8041.182} C_VEL
LIN {X 0,Y 462.021,Z 780.132,A -85,B 0,C 180,E1 -8043.726,E2 -8043.726} C_VEL
LIN {X 0,Y 462.288,Z 776.924,A -85,B 0,C 180,E1 -8045.289,E2 -8045.289} C_VEL
LIN {X 0,Y 462.29,Z 774.921,A -85,B 0,C 180,E1 -8046.363,E2 -8046.363} C_VEL
LIN {X 0,Y 461.792,Z 771.327,A -85,B 0,C 180,E1 -8048.607,E2 -8048.607} C_VEL
LIN {X 0,Y 461.314,Z 768.377,A -85,B 0,C 180,E1 -8050.927,E2 -8050.927} C_VEL
LIN {X 0,Y 460.883,Z 766.185,A -85,B 0,C 180,E1 -8053.331,E2 -8053.331} C_VEL
LIN {X 0,Y 460.61,Z 764.814,A -85,B 0,C 180,E1 -8055.818,E2 -8055.818} C_VEL
LIN {X 0,Y 460.562,Z 764.27,A -85,B 0,C 180,E1 -8058.394,E2 -8058.394} C_VEL
LIN {X 0,Y 460.576,Z 764.535,A -85,B 0,C 180,E1 -8061.271,E2 -8061.271} C_VEL
LIN {X 0,Y 460.662,Z 765.426,A -85,B 0,C 180,E1 -8063.958,E2 -8063.958} C_VEL
LIN {X 0,Y 460.611,Z 766.991,A -85,B 0,C 180,E1 -8067.055,E2 -8067.055} C_VEL
LIN {X 0,Y 460.374,Z 768.711,A -85,B 0,C 180,E1 -8069.749,E2 -8069.749} C_VEL
LIN {X 0,Y 460.213,Z 770.842,A -85,B 0,C 180,E1 -8072.732,E2 -8072.732} C_VEL
LIN {X 0,Y 460.058,Z 773.107,A -85,B 0,C 180,E1 -8075.64,E2 -8075.64} C_VEL
LIN {X 0,Y 459.99,Z 775.694,A -85,B 0,C 180,E1 -8078.749,E2 -8078.749} C_VEL
LIN {X 0,Y 459.876,Z 777.981,A -85,B 0,C 180,E1 -8081.354,E2 -8081.354} C_VEL
LIN {X 0,Y 459.842,Z 781.036,A -85,B 0,C 180,E1 -8084.532,E2 -8084.532} C_VEL
LIN {X 0,Y 462.623,Z 792.767,A -85,B 0,C 180,E1 -8085.014,E2 -8085.014} C_VEL
LIN {X 0,Y 463.237,Z 798.516,A -85,B 0,C 180,E1 -8085.278,E2 -8085.278} C_VEL
LIN {X 0,Y 462.788,Z 811.246,A -85,B 0,C 180,E1 -8085.937,E2 -8085.937} C_VEL
LIN {X 0,Y 462.346,Z 822.596,A -85,B 0,C 180,E1 -8086.712,E2 -8086.712} C_VEL
LIN {X 0,Y 461.817,Z 833.992,A -85,B 0,C 180,E1 -8087.698,E2 -8087.698} C_VEL
LIN {X 0,Y 461.22,Z 844.195,A -85,B 0,C 180,E1 -8088.796,E2 -8088.796} C_VEL
LIN {X 0,Y 460.867,Z 852.464,A -85,B 0,C 180,E1 -8089.899,E2 -8089.899} C_VEL
LIN {X 0,Y 460.416,Z 860.56,A -85,B 0,C 180,E1 -8091.219,E2 -8091.219} C_VEL
LIN {X 0,Y 460.107,Z 867.061,A -85,B 0,C 180,E1 -8092.539,E2 -8092.539} C_VEL
LIN {X 0,Y 459.967,Z 872.213,A -85,B 0,C 180,E1 -8093.859,E2 -8093.859} C_VEL
LIN {X 0,Y 459.763,Z 876.203,A -85,B 0,C 180,E1 -8095.176,E2 -8095.176} C_VEL
LIN {X 0,Y 459.704,Z 879.133,A -85,B 0,C 180,E1 -8096.493,E2 -8096.493} C_VEL
LIN {X 0,Y 459.656,Z 880.546,A -85,B 0,C 180,E1 -8097.37,E2 -8097.37} C_VEL
LIN {X 0,Y 459.628,Z 881.534,A -85,B 0,C 180,E1 -8098.247,E2 -8098.247} C_VEL
LIN {X 0,Y 459.53,Z 882.355,A -85,B 0,C 180,E1 -8099.999,E2 -8099.999} C_VEL
LIN {X 0,Y 459.553,Z 882.146,A -85,B 0,C 180,E1 -8100.875,E2 -8100.875} C_VEL
LIN {X 0,Y 459.626,Z 881.53,A -85,B 0,C 180,E1 -8101.752,E2 -8101.752} C_VEL
LIN {X 0,Y 459.701,Z 879.134,A -85,B 0,C 180,E1 -8103.505,E2 -8103.505} C_VEL
LIN {X 0,Y 459.697,Z 876.208,A -85,B 0,C 180,E1 -8104.823,E2 -8104.823} C_VEL
LIN {X 0,Y 459.944,Z 872.235,A -85,B 0,C 180,E1 -8106.139,E2 -8106.139} C_VEL
LIN {X 0,Y 460.096,Z 866.126,A -85,B 0,C 180,E1 -8107.68,E2 -8107.68} C_VEL
LIN {X 0,Y 460.436,Z 859.441,A -85,B 0,C 180,E1 -8109,E2 -8109} C_VEL
LIN {X 0,Y 460.843,Z 851.143,A -85,B 0,C 180,E1 -8110.322,E2 -8110.322} C_VEL
LIN {X 0,Y 461.256,Z 842.615,A -85,B 0,C 180,E1 -8111.424,E2 -8111.424} C_VEL
LIN {X 0,Y 461.833,Z 832.311,A -85,B 0,C 180,E1 -8112.503,E2 -8112.503} C_VEL
LIN {X 0,Y 462.259,Z 821.296,A -85,B 0,C 180,E1 -8113.438,E2 -8113.438} C_VEL
LIN {X 0,Y 462.741,Z 810.346,A -85,B 0,C 180,E1 -8114.175,E2 -8114.175} C_VEL
LIN {X 0,Y 463.164,Z 797.433,A -85,B 0,C 180,E1 -8114.835,E2 -8114.835} C_VEL
LIN {X 0,Y 461.685,Z 788.055,A -85,B 0,C 180,E1 -8115.255,E2 -8115.255} C_VEL
LIN {X 0,Y 459.661,Z 779.239,A -85,B 0,C 180,E1 -8115.6,E2 -8115.6} C_VEL
LIN {X 0,Y 459.652,Z 775.929,A -85,B 0,C 180,E1 -8118.728,E2 -8118.728} C_VEL
LIN {X 0,Y 459.729,Z 773.02,A -85,B 0,C 180,E1 -8121.523,E2 -8121.523} C_VEL
LIN {X 0,Y 459.786,Z 770.068,A -85,B 0,C 180,E1 -8124.374,E2 -8124.374} C_VEL
LIN {X 0,Y 459.86,Z 766.826,A -85,B 0,C 180,E1 -8127.574,E2 -8127.574} C_VEL
LIN {X 0,Y 459.898,Z 764.201,A -85,B 0,C 180,E1 -8130.283,E2 -8130.283} C_VEL
LIN {X 0,Y 460.235,Z 764.156,A -85,B 0,C 180,E1 -8133.348,E2 -8133.348} C_VEL
LIN {X 0,Y 460.448,Z 764.128,A -85,B 0,C 180,E1 -8136.005,E2 -8136.005} C_VEL
LIN {X 0,Y 460.539,Z 764.12,A -85,B 0,C 180,E1 -8138.896,E2 -8138.896} C_VEL
LIN {X 0,Y 460.518,Z 764.119,A -85,B 0,C 180,E1 -8142.18,E2 -8142.18} C_VEL
LIN {X 0,Y 460.512,Z 764.122,A -85,B 0,C 180,E1 -8145.411,E2 -8145.411} C_VEL
LIN {X 0,Y 460.526,Z 764.117,A -85,B 0,C 180,E1 -8148.397,E2 -8148.397} C_VEL
LIN {X 0,Y 460.517,Z 764.124,A -85,B 0,C 180,E1 -8151.266,E2 -8151.266} C_VEL
LIN {X 0,Y 460.501,Z 764.12,A -85,B 0,C 180,E1 -8154.553,E2 -8154.553} C_VEL
LIN {X 0,Y 460.522,Z 764.12,A -85,B 0,C 180,E1 -8157.715,E2 -8157.715} C_VEL
LIN {X 0,Y 460.519,Z 764.118,A -85,B 0,C 180,E1 -8160.767,E2 -8160.767} C_VEL
LIN {X 0,Y 460.522,Z 764.121,A -85,B 0,C 180,E1 -8163.732,E2 -8163.732} C_VEL
LIN {X 0,Y 460.535,Z 764.115,A -85,B 0,C 180,E1 -8166.623,E2 -8166.623} C_VEL
LIN {X 0,Y 460.542,Z 764.119,A -85,B 0,C 180,E1 -8169.452,E2 -8169.452} C_VEL
LIN {X 0,Y 460.537,Z 764.116,A -85,B 0,C 180,E1 -8172.229,E2 -8172.229} C_VEL
LIN {X 0,Y 460.554,Z 764.113,A -85,B 0,C 180,E1 -8174.964,E2 -8174.964} C_VEL
LIN {X 0,Y 460.539,Z 764.115,A -85,B 0,C 180,E1 -8175.226,E2 -8175.226} C_VEL
LIN {X 0,Y 459.861,Z 764.204,A -85,B 0,C 180,E1 -8175.956,E2 -8175.956} C_VEL
LIN {X 0,Y 457.013,Z 764.554,A -85,B 0,C 180,E1 -8177.142,E2 -8177.142} C_VEL
LIN {X 0,Y 454.616,Z 764.856,A -85,B 0,C 180,E1 -8178.099,E2 -8178.099} C_VEL
LIN {X 0,Y 453.593,Z 764.98,A -85,B 0,C 180,E1 -8178.838,E2 -8178.838} C_VEL
LIN {X 0,Y 453.512,Z 764.99,A -85,B 0,C 180,E1 -8179.088,E2 -8179.088} C_VEL
LIN {X 0,Y 453.619,Z 764.977,A -85,B 0,C 180,E1 -8182.542,E2 -8182.542} C_VEL
LIN {X 0,Y 453.636,Z 764.974,A -85,B 0,C 180,E1 -8184.666,E2 -8184.666} C_VEL
LIN {X 0,Y 453.675,Z 764.973,A -85,B 0,C 180,E1 -8188.225,E2 -8188.225} C_VEL
LIN {X 0,Y 453.756,Z 764.966,A -85,B 0,C 180,E1 -8190,E2 -8190} C_VEL
LIN {X 0,Y 453.689,Z 764.968,A -85,B 0,C 180,E1 -8192.664,E2 -8192.664} C_VEL
LIN {X 0,Y 453.623,Z 764.982,A -85,B 0,C 180,E1 -8196.226,E2 -8196.226} C_VEL
LIN {X 0,Y 453.544,Z 764.985,A -85,B 0,C 180,E1 -8198.914,E2 -8198.914} C_VEL
LIN {X 0,Y 453.554,Z 764.988,A -85,B 0,C 180,E1 -8202.529,E2 -8202.529} C_VEL
LIN {X 0,Y 453.535,Z 764.992,A -85,B 0,C 180,E1 -8206.196,E2 -8206.196} C_VEL
LIN {X 0,Y 453.507,Z 764.991,A -85,B 0,C 180,E1 -8209.04,E2 -8209.04} C_VEL
LIN {X 0,Y 453.467,Z 764.997,A -85,B 0,C 180,E1 -8211.837,E2 -8211.837} C_VEL
LIN {X 0,Y 453.481,Z 764.998,A -85,B 0,C 180,E1 -8214.736,E2 -8214.736} C_VEL
LIN {X 0,Y 453.481,Z 764.995,A -85,B 0,C 180,E1 -8217.95,E2 -8217.95} C_VEL
LIN {X 0,Y 453.467,Z 765.001,A -85,B 0,C 180,E1 -8220.76,E2 -8220.76} C_VEL
LIN {X 0,Y 453.461,Z 764.998,A -85,B 0,C 180,E1 -8223.914,E2 -8223.914} C_VEL
LIN {X 0,Y 453.445,Z 765.001,A -85,B 0,C 180,E1 -8227.191,E2 -8227.191} C_VEL
LIN {X 0,Y 453.479,Z 764.995,A -85,B 0,C 180,E1 -8229.451,E2 -8229.451} C_VEL
LIN {X 0,Y 453.47,Z 764.997,A -85,B 0,C 180,E1 -8231.936,E2 -8231.936} C_VEL
LIN {X 0,Y 453.479,Z 764.996,A -85,B 0,C 180,E1 -8235.472,E2 -8235.472} C_VEL
LIN {X 0,Y 453.474,Z 764.997,A -85,B 0,C 180,E1 -8238.21,E2 -8238.21} C_VEL
LIN {X 0,Y 453.49,Z 764.997,A -85,B 0,C 180,E1 -8240.794,E2 -8240.794} C_VEL
LIN {X 0,Y 453.416,Z 765.003,A -85,B 0,C 180,E1 -8243.915,E2 -8243.915} C_VEL
LIN {X 0,Y 453.235,Z 765.03,A -85,B 0,C 180,E1 -8247.132,E2 -8247.132} C_VEL
LIN {X 0,Y 452.77,Z 765.089,A -85,B 0,C 180,E1 -8250.372,E2 -8250.372} C_VEL
LIN {X 0,Y 452.663,Z 765.243,A -85,B 0,C 180,E1 -8251.231,E2 -8251.231} C_VEL
LIN {X 0,Y 452.716,Z 768.5,A -85,B 0,C 180,E1 -8254.237,E2 -8254.237} C_VEL
LIN {X 0,Y 452.62,Z 771.703,A -85,B 0,C 180,E1 -8257.16,E2 -8257.16} C_VEL
LIN {X 0,Y 452.619,Z 774.812,A -85,B 0,C 180,E1 -8260.027,E2 -8260.027} C_VEL
LIN {X 0,Y 452.544,Z 777.896,A -85,B 0,C 180,E1 -8262.839,E2 -8262.839} C_VEL
LIN {X 0,Y 452.578,Z 779.448,A -85,B 0,C 180,E1 -8264.277,E2 -8264.277} C_VEL
LIN {X 0,Y 455.448,Z 792.443,A -85,B 0,C 180,E1 -8264.793,E2 -8264.793} C_VEL
LIN {X 0,Y 456.258,Z 798.999,A -85,B 0,C 180,E1 -8265.106,E2 -8265.106} C_VEL
LIN {X 0,Y 455.782,Z 811.589,A -85,B 0,C 180,E1 -8265.781,E2 -8265.781} C_VEL
LIN {X 0,Y 455.247,Z 823.432,A -85,B 0,C 180,E1 -8266.612,E2 -8266.612} C_VEL
LIN {X 0,Y 454.776,Z 834.668,A -85,B 0,C 180,E1 -8267.619,E2 -8267.619} C_VEL
LIN {X 0,Y 454.204,Z 843.818,A -85,B 0,C 180,E1 -8268.623,E2 -8268.623} C_VEL
LIN {X 0,Y 453.817,Z 852.21,A -85,B 0,C 180,E1 -8269.742,E2 -8269.742} C_VEL
LIN {X 0,Y 453.363,Z 860.367,A -85,B 0,C 180,E1 -8271.083,E2 -8271.083} C_VEL
LIN {X 0,Y 453.022,Z 866.944,A -85,B 0,C 180,E1 -8272.424,E2 -8272.424} C_VEL
LIN {X 0,Y 452.886,Z 872.181,A -85,B 0,C 180,E1 -8273.765,E2 -8273.765} C_VEL
LIN {X 0,Y 452.629,Z 876.255,A -85,B 0,C 180,E1 -8275.102,E2 -8275.102} C_VEL
LIN {X 0,Y 452.634,Z 879.263,A -85,B 0,C 180,E1 -8276.44,E2 -8276.44} C_VEL
LIN {X 0,Y 452.532,Z 880.738,A -85,B 0,C 180,E1 -8277.33,E2 -8277.33} C_VEL
LIN {X 0,Y 452.562,Z 881.769,A -85,B 0,C 180,E1 -8278.221,E2 -8278.221} C_VEL
LIN {X 0,Y 452.464,Z 882.691,A -85,B 0,C 180,E1 -8280.001,E2 -8280.001} C_VEL
LIN {X 0,Y 452.489,Z 882.517,A -85,B 0,C 180,E1 -8280.891,E2 -8280.891} C_VEL
LIN {X 0,Y 452.565,Z 881.945,A -85,B 0,C 180,E1 -8281.781,E2 -8281.781} C_VEL
LIN {X 0,Y 452.554,Z 880.994,A -85,B 0,C 180,E1 -8282.671,E2 -8282.671} C_VEL
LIN {X 0,Y 452.642,Z 879.622,A -85,B 0,C 180,E1 -8283.562,E2 -8283.562} C_VEL
LIN {X 0,Y 452.672,Z 876.748,A -85,B 0,C 180,E1 -8284.899,E2 -8284.899} C_VEL
LIN {X 0,Y 452.922,Z 872.817,A -85,B 0,C 180,E1 -8286.237,E2 -8286.237} C_VEL
LIN {X 0,Y 453.044,Z 867.726,A -85,B 0,C 180,E1 -8287.578,E2 -8287.578} C_VEL
LIN {X 0,Y 453.395,Z 861.297,A -85,B 0,C 180,E1 -8288.918,E2 -8288.918} C_VEL
LIN {X 0,Y 453.841,Z 853.31,A -85,B 0,C 180,E1 -8290.259,E2 -8290.259} C_VEL
LIN {X 0,Y 454.247,Z 845.118,A -85,B 0,C 180,E1 -8291.378,E2 -8291.378} C_VEL
LIN {X 0,Y 454.877,Z 835.018,A -85,B 0,C 180,E1 -8292.493,E2 -8292.493} C_VEL
LIN {X 0,Y 455.227,Z 824.578,A -85,B 0,C 180,E1 -8293.437,E2 -8293.437} C_VEL
LIN {X 0,Y 455.847,Z 812.633,A -85,B 0,C 180,E1 -8294.282,E2 -8294.282} C_VEL
LIN {X 0,Y 456.347,Z 799.166,A -85,B 0,C 180,E1 -8295.007,E2 -8295.007} C_VEL
LIN {X 0,Y 455.195,Z 790.928,A -85,B 0,C 180,E1 -8295.395,E2 -8295.395} C_VEL
LIN {X 0,Y 452.691,Z 780.92,A -85,B 0,C 180,E1 -8295.835,E2 -8295.835} C_VEL
LIN {X 0,Y 452.724,Z 777.456,A -85,B 0,C 180,E1 -8299.027,E2 -8299.027} C_VEL
LIN {X 0,Y 452.721,Z 774.288,A -85,B 0,C 180,E1 -8301.875,E2 -8301.875} C_VEL
LIN {X 0,Y 452.771,Z 770.984,A -85,B 0,C 180,E1 -8304.779,E2 -8304.779} C_VEL
LIN {X 0,Y 452.779,Z 767.375,A -85,B 0,C 180,E1 -8307.779,E2 -8307.779} C_VEL
LIN {X 0,Y 452.792,Z 765.088,A -85,B 0,C 180,E1 -8309.782,E2 -8309.782} C_VEL
LIN {X 0,Y 453.207,Z 765.035,A -85,B 0,C 180,E1 -8313.134,E2 -8313.134} C_VEL
LIN {X 0,Y 453.42,Z 765.004,A -85,B 0,C 180,E1 -8316.087,E2 -8316.087} C_VEL
LIN {X 0,Y 453.473,Z 765.001,A -85,B 0,C 180,E1 -8319.203,E2 -8319.203} C_VEL
LIN {X 0,Y 453.464,Z 764.998,A -85,B 0,C 180,E1 -8321.933,E2 -8321.933} C_VEL
LIN {X 0,Y 453.492,Z 764.997,A -85,B 0,C 180,E1 -8325.471,E2 -8325.471} C_VEL
LIN {X 0,Y 453.504,Z 765.009,A -85,B 0,C 180,E1 -8328.657,E2 -8328.657} C_VEL
LIN {X 0,Y 454.72,Z 771.812,A -85,B 0,C 180,E1 -8331.813,E2 -8331.813} C_VEL
LIN {X 0,Y 455.409,Z 776.993,A -85,B 0,C 180,E1 -8334.096,E2 -8334.096} C_VEL
LIN {X 0,Y 455.014,Z 784.754,A -85,B 0,C 180,E1 -8337.275,E2 -8337.275} C_VEL
LIN {X 0,Y 454.493,Z 792.515,A -85,B 0,C 180,E1 -8340.341,E2 -8340.341} C_VEL
LIN {X 0,Y 454.108,Z 800.311,A -85,B 0,C 180,E1 -8343.332,E2 -8343.332} C_VEL
LIN {X 0,Y 453.711,Z 808.142,A -85,B 0,C 180,E1 -8346.25,E2 -8346.25} C_VEL
LIN {X 0,Y 453.362,Z 817.294,A -85,B 0,C 180,E1 -8349.586,E2 -8349.586} C_VEL
LIN {X 0,Y 453.045,Z 826.475,A -85,B 0,C 180,E1 -8352.858,E2 -8352.858} C_VEL
LIN {X 0,Y 452.985,Z 830.177,A -85,B 0,C 180,E1 -8354.139,E2 -8354.139} C_VEL
LIN {X 0,Y 454.976,Z 843.788,A -85,B 0,C 180,E1 -8354.593,E2 -8354.593} C_VEL
LIN {X 0,Y 456.122,Z 852.524,A -85,B 0,C 180,E1 -8354.986,E2 -8354.986} C_VEL
LIN {X 0,Y 455.617,Z 864.381,A -85,B 0,C 180,E1 -8355.597,E2 -8355.597} C_VEL
LIN {X 0,Y 455.043,Z 875.986,A -85,B 0,C 180,E1 -8356.377,E2 -8356.377} C_VEL
LIN {X 0,Y 454.512,Z 887.355,A -85,B 0,C 180,E1 -8357.351,E2 -8357.351} C_VEL
LIN {X 0,Y 454.016,Z 897.177,A -85,B 0,C 180,E1 -8358.391,E2 -8358.391} C_VEL
LIN {X 0,Y 453.533,Z 905.858,A -85,B 0,C 180,E1 -8359.509,E2 -8359.509} C_VEL
LIN {X 0,Y 453.125,Z 914.297,A -85,B 0,C 180,E1 -8360.852,E2 -8360.852} C_VEL
LIN {X 0,Y 452.83,Z 921.097,A -85,B 0,C 180,E1 -8362.195,E2 -8362.195} C_VEL
LIN {X 0,Y 452.634,Z 927.339,A -85,B 0,C 180,E1 -8363.76,E2 -8363.76} C_VEL
LIN {X 0,Y 452.569,Z 931.384,A -85,B 0,C 180,E1 -8365.1,E2 -8365.1} C_VEL
LIN {X 0,Y 452.525,Z 934.363,A -85,B 0,C 180,E1 -8366.438,E2 -8366.438} C_VEL
LIN {X 0,Y 452.5,Z 935.785,A -85,B 0,C 180,E1 -8367.329,E2 -8367.329} C_VEL
LIN {X 0,Y 452.527,Z 936.789,A -85,B 0,C 180,E1 -8368.22,E2 -8368.22} C_VEL
LIN {X 0,Y 452.489,Z 937.391,A -85,B 0,C 180,E1 -8369.11,E2 -8369.11} C_VEL
LIN {X 0,Y 452.464,Z 937.592,A -85,B 0,C 180,E1 -8370,E2 -8370} C_VEL
LIN {X 0,Y 452.489,Z 937.353,A -85,B 0,C 180,E1 -8370.89,E2 -8370.89} C_VEL
LIN {X 0,Y 452.527,Z 936.706,A -85,B 0,C 180,E1 -8371.78,E2 -8371.78} C_VEL
LIN {X 0,Y 452.502,Z 935.653,A -85,B 0,C 180,E1 -8372.671,E2 -8372.671} C_VEL
LIN {X 0,Y 452.555,Z 934.189,A -85,B 0,C 180,E1 -8373.561,E2 -8373.561} C_VEL
LIN {X 0,Y 452.57,Z 931.124,A -85,B 0,C 180,E1 -8374.9,E2 -8374.9} C_VEL
LIN {X 0,Y 452.652,Z 926.248,A -85,B 0,C 180,E1 -8376.441,E2 -8376.441} C_VEL
LIN {X 0,Y 452.875,Z 919.576,A -85,B 0,C 180,E1 -8378.029,E2 -8378.029} C_VEL
LIN {X 0,Y 453.179,Z 912.4,A -85,B 0,C 180,E1 -8379.372,E2 -8379.372} C_VEL
LIN {X 0,Y 453.566,Z 903.425,A -85,B 0,C 180,E1 -8380.716,E2 -8380.716} C_VEL
LIN {X 0,Y 454.103,Z 893.274,A -85,B 0,C 180,E1 -8381.947,E2 -8381.947} C_VEL
LIN {X 0,Y 454.618,Z 882.984,A -85,B 0,C 180,E1 -8382.952,E2 -8382.952} C_VEL
LIN {X 0,Y 455.142,Z 871.621,A -85,B 0,C 180,E1 -8383.848,E2 -8383.848} C_VEL
LIN {X 0,Y 455.758,Z 859.031,A -85,B 0,C 180,E1 -8384.626,E2 -8384.626} C_VEL
LIN {X 0,Y 455.934,Z 850.967,A -85,B 0,C 180,E1 -8385.02,E2 -8385.02} C_VEL
LIN {X 0,Y 454.176,Z 837.878,A -85,B 0,C 180,E1 -8385.579,E2 -8385.579} C_VEL
LIN {X 0,Y 452.935,Z 828.5,A -85,B 0,C 180,E1 -8385.89,E2 -8385.89} C_VEL
LIN {X 0,Y 453.107,Z 819.37,A -85,B 0,C 180,E1 -8389.01,E2 -8389.01} C_VEL
LIN {X 0,Y 453.392,Z 809.947,A -85,B 0,C 180,E1 -8392.32,E2 -8392.32} C_VEL
LIN {X 0,Y 453.732,Z 800.701,A -85,B 0,C 180,E1 -8395.703,E2 -8395.703} C_VEL
LIN {X 0,Y 454.109,Z 793.073,A -85,B 0,C 180,E1 -8398.671,E2 -8398.671} C_VEL
LIN {X 0,Y 454.714,Z 784.671,A -85,B 0,C 180,E1 -8402.223,E2 -8402.223} C_VEL
LIN {X 0,Y 455.209,Z 779.188,A -85,B 0,C 180,E1 -8404.837,E2 -8404.837} C_VEL
LIN {X 0,Y 455.281,Z 775.922,A -85,B 0,C 180,E1 -8406.61,E2 -8406.61} C_VEL
LIN {X 0,Y 454.675,Z 771.858,A -85,B 0,C 180,E1 -8409.327,E2 -8409.327} C_VEL
LIN {X 0,Y 454.174,Z 768.823,A -85,B 0,C 180,E1 -8412.032,E2 -8412.032} C_VEL
LIN {X 0,Y 453.831,Z 766.937,A -85,B 0,C 180,E1 -8414.572,E2 -8414.572} C_VEL
LIN {X 0,Y 453.622,Z 765.965,A -85,B 0,C 180,E1 -8417.023,E2 -8417.023} C_VEL
LIN {X 0,Y 453.599,Z 765.708,A -85,B 0,C 180,E1 -8419.402,E2 -8419.402} C_VEL
LIN {X 0,Y 453.64,Z 766.131,A -85,B 0,C 180,E1 -8422.197,E2 -8422.197} C_VEL
LIN {X 0,Y 453.667,Z 767.22,A -85,B 0,C 180,E1 -8425.191,E2 -8425.191} C_VEL
LIN {X 0,Y 453.488,Z 768.836,A -85,B 0,C 180,E1 -8428.202,E2 -8428.202} C_VEL
LIN {X 0,Y 453.262,Z 770.83,A -85,B 0,C 180,E1 -8431.27,E2 -8431.27} C_VEL
LIN {X 0,Y 453.111,Z 772.994,A -85,B 0,C 180,E1 -8434.259,E2 -8434.259} C_VEL
LIN {X 0,Y 452.995,Z 775.296,A -85,B 0,C 180,E1 -8437.178,E2 -8437.178} C_VEL
LIN {X 0,Y 452.876,Z 777.694,A -85,B 0,C 180,E1 -8440.036,E2 -8440.036} C_VEL
LIN {X 0,Y 452.731,Z 780.177,A -85,B 0,C 180,E1 -8442.845,E2 -8442.845} C_VEL
LIN {X 0,Y 452.779,Z 781.464,A -85,B 0,C 180,E1 -8444.266,E2 -8444.266} C_VEL
LIN {X 0,Y 455.837,Z 794.068,A -85,B 0,C 180,E1 -8444.819,E2 -8444.819} C_VEL
LIN {X 0,Y 456.403,Z 798.903,A -85,B 0,C 180,E1 -8445.052,E2 -8445.052} C_VEL
LIN {X 0,Y 455.935,Z 811.615,A -85,B 0,C 180,E1 -8445.721,E2 -8445.721} C_VEL
LIN {X 0,Y 455.446,Z 823.061,A -85,B 0,C 180,E1 -8446.514,E2 -8446.514} C_VEL
LIN {X 0,Y 454.906,Z 834.383,A -85,B 0,C 180,E1 -8447.508,E2 -8447.508} C_VEL
LIN {X 0,Y 454.273,Z 844.606,A -85,B 0,C 180,E1 -8448.623,E2 -8448.623} C_VEL
LIN {X 0,Y 453.782,Z 854.358,A -85,B 0,C 180,E1 -8449.965,E2 -8449.965} C_VEL
LIN {X 0,Y 453.358,Z 862.197,A -85,B 0,C 180,E1 -8451.306,E2 -8451.306} C_VEL
LIN {X 0,Y 453.067,Z 867.486,A -85,B 0,C 180,E1 -8452.422,E2 -8452.422} C_VEL
LIN {X 0,Y 452.931,Z 872.639,A -85,B 0,C 180,E1 -8453.764,E2 -8453.764} C_VEL
LIN {X 0,Y 452.703,Z 876.633,A -85,B 0,C 180,E1 -8455.101,E2 -8455.101} C_VEL
LIN {X 0,Y 452.645,Z 879.565,A -85,B 0,C 180,E1 -8456.438,E2 -8456.438} C_VEL
LIN {X 0,Y 452.578,Z 880.983,A -85,B 0,C 180,E1 -8457.329,E2 -8457.329} C_VEL
LIN {X 0,Y 452.568,Z 881.968,A -85,B 0,C 180,E1 -8458.219,E2 -8458.219} C_VEL
LIN {X 0,Y 452.464,Z 882.785,A -85,B 0,C 180,E1 -8459.999,E2 -8459.999} C_VEL
LIN {X 0,Y 452.489,Z 882.571,A -85,B 0,C 180,E1 -8460.889,E2 -8460.889} C_VEL
LIN {X 0,Y 452.564,Z 881.948,A -85,B 0,C 180,E1 -8461.779,E2 -8461.779} C_VEL
LIN {X 0,Y 452.638,Z 879.536,A -85,B 0,C 180,E1 -8463.56,E2 -8463.56} C_VEL
LIN {X 0,Y 452.623,Z 876.595,A -85,B 0,C 180,E1 -8464.898,E2 -8464.898} C_VEL
LIN {X 0,Y 452.894,Z 872.602,A -85,B 0,C 180,E1 -8466.235,E2 -8466.235} C_VEL
LIN {X 0,Y 453.052,Z 866.466,A -85,B 0,C 180,E1 -8467.8,E2 -8467.8} C_VEL
LIN {X 0,Y 453.423,Z 859.753,A -85,B 0,C 180,E1 -8469.141,E2 -8469.141} C_VEL
LIN {X 0,Y 453.863,Z 851.428,A -85,B 0,C 180,E1 -8470.482,E2 -8470.482} C_VEL
LIN {X 0,Y 454.308,Z 842.865,A -85,B 0,C 180,E1 -8471.601,E2 -8471.601} C_VEL
LIN {X 0,Y 454.887,Z 832.675,A -85,B 0,C 180,E1 -8472.683,E2 -8472.683} C_VEL
LIN {X 0,Y 455.34,Z 821.916,A -85,B 0,C 180,E1 -8473.612,E2 -8473.612} C_VEL
LIN {X 0,Y 455.851,Z 810.497,A -85,B 0,C 180,E1 -8474.394,E2 -8474.394} C_VEL
LIN {X 0,Y 456.242,Z 797.568,A -85,B 0,C 180,E1 -8475.066,E2 -8475.066} C_VEL
LIN {X 0,Y 454.551,Z 788.091,A -85,B 0,C 180,E1 -8475.502,E2 -8475.502} C_VEL
LIN {X 0,Y 452.587,Z 779.586,A -85,B 0,C 180,E1 -8475.84,E2 -8475.84} C_VEL
LIN {X 0,Y 452.591,Z 776.234,A -85,B 0,C 180,E1 -8479.031,E2 -8479.031} C_VEL
LIN {X 0,Y 452.661,Z 773.271,A -85,B 0,C 180,E1 -8481.876,E2 -8481.876} C_VEL
LIN {X 0,Y 452.721,Z 770.297,A -85,B 0,C 180,E1 -8484.779,E2 -8484.779} C_VEL
LIN {X 0,Y 452.773,Z 767.267,A -85,B 0,C 180,E1 -8487.777,E2 -8487.777} C_VEL
LIN {X 0,Y 452.807,Z 765.288,A -85,B 0,C 180,E1 -8489.779,E2 -8489.779} C_VEL
LIN {X 0,Y 453.166,Z 765.039,A -85,B 0,C 180,E1 -8492.873,E2 -8492.873} C_VEL
LIN {X 0,Y 453.371,Z 765.013,A -85,B 0,C 180,E1 -8494.998,E2 -8494.998} C_VEL
LIN {X 0,Y 453.459,Z 764.998,A -85,B 0,C 180,E1 -8498.311,E2 -8498.311} C_VEL
LIN {X 0,Y 453.49,Z 764.995,A -85,B 0,C 180,E1 -8500.608,E2 -8500.608} C_VEL
LIN {X 0,Y 453.451,Z 765.002,A -85,B 0,C 180,E1 -8503.243,E2 -8503.243} C_VEL
LIN {X 0,Y 453.461,Z 764.999,A -85,B 0,C 180,E1 -8505.778,E2 -8505.778} C_VEL
LIN {X 0,Y 453.473,Z 764.996,A -85,B 0,C 180,E1 -8508.208,E2 -8508.208} C_VEL
LIN {X 0,Y 453.485,Z 764.996,A -85,B 0,C 180,E1 -8510.793,E2 -8510.793} C_VEL
LIN {X 0,Y 453.447,Z 765.001,A -85,B 0,C 180,E1 -8513.916,E2 -8513.916} C_VEL
LIN {X 0,Y 453.471,Z 764.999,A -85,B 0,C 180,E1 -8517.15,E2 -8517.15} C_VEL
LIN {X 0,Y 453.459,Z 764.998,A -85,B 0,C 180,E1 -8520.267,E2 -8520.267} C_VEL
LIN {X 0,Y 453.463,Z 765.001,A -85,B 0,C 180,E1 -8523.291,E2 -8523.291} C_VEL
LIN {X 0,Y 453.484,Z 764.995,A -85,B 0,C 180,E1 -8526.238,E2 -8526.238} C_VEL
LIN {X 0,Y 453.473,Z 764.996,A -85,B 0,C 180,E1 -8529.117,E2 -8529.117} C_VEL
LIN {X 0,Y 453.492,Z 764.996,A -85,B 0,C 180,E1 -8531.944,E2 -8531.944} C_VEL
LIN {X 0,Y 453.529,Z 764.988,A -85,B 0,C 180,E1 -8534.726,E2 -8534.726} C_VEL
LIN {X 0,Y 453.548,Z 764.987,A -85,B 0,C 180,E1 -8538.379,E2 -8538.379} C_VEL
LIN {X 0,Y 453.512,Z 764.99,A -85,B 0,C 180,E1 -8539.088,E2 -8539.088} C_VEL
LIN {X 0,Y 452.859,Z 765.078,A -85,B 0,C 180,E1 -8539.829,E2 -8539.829} C_VEL
LIN {X 0,Y 450.04,Z 765.425,A -85,B 0,C 180,E1 -8541.034,E2 -8541.034} C_VEL
LIN {X 0,Y 447.656,Z 765.724,A -85,B 0,C 180,E1 -8542.006,E2 -8542.006} C_VEL
LIN {X 0,Y 446.64,Z 765.846,A -85,B 0,C 180,E1 -8542.756,E2 -8542.756} C_VEL
LIN {X 0,Y 446.561,Z 765.855,A -85,B 0,C 180,E1 -8543.01,E2 -8543.01} C_VEL
LIN {X 0,Y 446.61,Z 765.85,A -85,B 0,C 180,E1 -8544.582,E2 -8544.582} C_VEL
LIN {X 0,Y 446.645,Z 765.849,A -85,B 0,C 180,E1 -8548.197,E2 -8548.197} C_VEL
LIN {X 0,Y 446.707,Z 765.845,A -85,B 0,C 180,E1 -8550,E2 -8550} C_VEL
LIN {X 0,Y 446.638,Z 765.846,A -85,B 0,C 180,E1 -8552.706,E2 -8552.706} C_VEL
LIN {X 0,Y 446.593,Z 765.856,A -85,B 0,C 180,E1 -8556.324,E2 -8556.324} C_VEL
LIN {X 0,Y 446.495,Z 765.863,A -85,B 0,C 180,E1 -8559.056,E2 -8559.056} C_VEL
LIN {X 0,Y 446.512,Z 765.864,A -85,B 0,C 180,E1 -8562.73,E2 -8562.73} C_VEL
LIN {X 0,Y 446.478,Z 765.872,A -85,B 0,C 180,E1 -8566.46,E2 -8566.46} C_VEL
LIN {X 0,Y 446.459,Z 765.868,A -85,B 0,C 180,E1 -8569.304,E2 -8569.304} C_VEL
LIN {X 0,Y 446.409,Z 765.878,A -85,B 0,C 180,E1 -8572.2,E2 -8572.2} C_VEL
LIN {X 0,Y 446.423,Z 765.874,A -85,B 0,C 180,E1 -8575.155,E2 -8575.155} C_VEL
LIN {X 0,Y 446.432,Z 765.874,A -85,B 0,C 180,E1 -8578.182,E2 -8578.182} C_VEL
LIN {X 0,Y 446.407,Z 765.876,A -85,B 0,C 180,E1 -8581.301,E2 -8581.301} C_VEL
LIN {X 0,Y 446.415,Z 765.878,A -85,B 0,C 180,E1 -8584.524,E2 -8584.524} C_VEL
LIN {X 0,Y 446.408,Z 765.877,A -85,B 0,C 180,E1 -8588.08,E2 -8588.08} C_VEL
LIN {X 0,Y 446.421,Z 765.879,A -85,B 0,C 180,E1 -8590.919,E2 -8590.919} C_VEL
LIN {X 0,Y 446.394,Z 765.878,A -85,B 0,C 180,E1 -8593.847,E2 -8593.847} C_VEL
LIN {X 0,Y 446.393,Z 765.879,A -85,B 0,C 180,E1 -8596.404,E2 -8596.404} C_VEL
LIN {X 0,Y 446.423,Z 765.879,A -85,B 0,C 180,E1 -8599.083,E2 -8599.083} C_VEL
LIN {X 0,Y 446.405,Z 765.878,A -85,B 0,C 180,E1 -8602.122,E2 -8602.122} C_VEL
LIN {X 0,Y 446.33,Z 765.889,A -85,B 0,C 180,E1 -8604.965,E2 -8604.965} C_VEL
LIN {X 0,Y 446.11,Z 765.919,A -85,B 0,C 180,E1 -8607.614,E2 -8607.614} C_VEL
LIN {X 0,Y 445.659,Z 765.975,A -85,B 0,C 180,E1 -8610.735,E2 -8610.735} C_VEL
LIN {X 0,Y 445.616,Z 766.726,A -85,B 0,C 180,E1 -8612.031,E2 -8612.031} C_VEL
LIN {X 0,Y 445.581,Z 769.718,A -85,B 0,C 180,E1 -8614.796,E2 -8614.796} C_VEL
LIN {X 0,Y 445.551,Z 772.942,A -85,B 0,C 180,E1 -8617.756,E2 -8617.756} C_VEL
LIN {X 0,Y 445.531,Z 776.096,A -85,B 0,C 180,E1 -8620.656,E2 -8620.656} C_VEL
LIN {X 0,Y 445.514,Z 779.895,A -85,B 0,C 180,E1 -8624.04,E2 -8624.04} C_VEL
LIN {X 0,Y 448.366,Z 792.343,A -85,B 0,C 180,E1 -8624.547,E2 -8624.547} C_VEL
LIN {X 0,Y 449.394,Z 798.997,A -85,B 0,C 180,E1 -8624.873,E2 -8624.873} C_VEL
LIN {X 0,Y 448.923,Z 810.623,A -85,B 0,C 180,E1 -8625.495,E2 -8625.495} C_VEL
LIN {X 0,Y 448.389,Z 822.27,A -85,B 0,C 180,E1 -8626.299,E2 -8626.299} C_VEL
LIN {X 0,Y 447.884,Z 833.704,A -85,B 0,C 180,E1 -8627.311,E2 -8627.311} C_VEL
LIN {X 0,Y 447.258,Z 844.025,A -85,B 0,C 180,E1 -8628.444,E2 -8628.444} C_VEL
LIN {X 0,Y 446.817,Z 852.461,A -85,B 0,C 180,E1 -8629.58,E2 -8629.58} C_VEL
LIN {X 0,Y 446.355,Z 860.656,A -85,B 0,C 180,E1 -8630.942,E2 -8630.942} C_VEL
LIN {X 0,Y 445.979,Z 867.261,A -85,B 0,C 180,E1 -8632.303,E2 -8632.303} C_VEL
LIN {X 0,Y 445.84,Z 872.523,A -85,B 0,C 180,E1 -8633.666,E2 -8633.666} C_VEL
LIN {X 0,Y 445.561,Z 876.62,A -85,B 0,C 180,E1 -8635.024,E2 -8635.024} C_VEL
LIN {X 0,Y 445.572,Z 879.645,A -85,B 0,C 180,E1 -8636.384,E2 -8636.384} C_VEL
LIN {X 0,Y 445.462,Z 881.134,A -85,B 0,C 180,E1 -8637.288,E2 -8637.288} C_VEL
LIN {X 0,Y 445.502,Z 882.174,A -85,B 0,C 180,E1 -8638.193,E2 -8638.193} C_VEL
LIN {X 0,Y 445.4,Z 883.108,A -85,B 0,C 180,E1 -8640.001,E2 -8640.001} C_VEL
LIN {X 0,Y 445.427,Z 882.94,A -85,B 0,C 180,E1 -8640.905,E2 -8640.905} C_VEL
LIN {X 0,Y 445.506,Z 882.371,A -85,B 0,C 180,E1 -8641.809,E2 -8641.809} C_VEL
LIN {X 0,Y 445.482,Z 881.423,A -85,B 0,C 180,E1 -8642.714,E2 -8642.714} C_VEL
LIN {X 0,Y 445.582,Z 880.053,A -85,B 0,C 180,E1 -8643.618,E2 -8643.618} C_VEL
LIN {X 0,Y 445.599,Z 877.181,A -85,B 0,C 180,E1 -8644.977,E2 -8644.977} C_VEL
LIN {X 0,Y 445.878,Z 873.243,A -85,B 0,C 180,E1 -8646.336,E2 -8646.336} C_VEL
LIN {X 0,Y 446.031,Z 868.142,A -85,B 0,C 180,E1 -8647.698,E2 -8647.698} C_VEL
LIN {X 0,Y 446.378,Z 861.703,A -85,B 0,C 180,E1 -8649.059,E2 -8649.059} C_VEL
LIN {X 0,Y 446.87,Z 853.7,A -85,B 0,C 180,E1 -8650.421,E2 -8650.421} C_VEL
LIN {X 0,Y 447.311,Z 845.485,A -85,B 0,C 180,E1 -8651.557,E2 -8651.557} C_VEL
LIN {X 0,Y 447.961,Z 835.403,A -85,B 0,C 180,E1 -8652.689,E2 -8652.689} C_VEL
LIN {X 0,Y 448.411,Z 824.203,A -85,B 0,C 180,E1 -8653.714,E2 -8653.714} C_VEL
LIN {X 0,Y 449.003,Z 813.139,A -85,B 0,C 180,E1 -8654.504,E2 -8654.504} C_VEL
LIN {X 0,Y 449.538,Z 799.821,A -85,B 0,C 180,E1 -8655.24,E2 -8655.24} C_VEL
LIN {X 0,Y 448.199,Z 791.437,A -85,B 0,C 180,E1 -8655.651,E2 -8655.651} C_VEL
LIN {X 0,Y 445.65,Z 781.424,A -85,B 0,C 180,E1 -8656.113,E2 -8656.113} C_VEL
LIN {X 0,Y 445.658,Z 777.921,A -85,B 0,C 180,E1 -8659.341,E2 -8659.341} C_VEL
LIN {X 0,Y 445.669,Z 774.721,A -85,B 0,C 180,E1 -8662.24,E2 -8662.24} C_VEL
LIN {X 0,Y 445.703,Z 771.29,A -85,B 0,C 180,E1 -8665.199,E2 -8665.199} C_VEL
LIN {X 0,Y 445.724,Z 767.762,A -85,B 0,C 180,E1 -8668.232,E2 -8668.232} C_VEL
LIN {X 0,Y 445.751,Z 765.965,A -85,B 0,C 180,E1 -8669.869,E2 -8669.869} C_VEL
LIN {X 0,Y 446.074,Z 765.924,A -85,B 0,C 180,E1 -8672.391,E2 -8672.391} C_VEL
LIN {X 0,Y 446.351,Z 765.887,A -85,B 0,C 180,E1 -8675.633,E2 -8675.633} C_VEL
LIN {X 0,Y 446.428,Z 765.88,A -85,B 0,C 180,E1 -8679.029,E2 -8679.029} C_VEL
LIN {X 0,Y 446.426,Z 765.875,A -85,B 0,C 180,E1 -8682.276,E2 -8682.276} C_VEL
LIN {X 0,Y 446.458,Z 765.875,A -85,B 0,C 180,E1 -8685.104,E2 -8685.104} C_VEL
LIN {X 0,Y 446.501,Z 766.079,A -85,B 0,C 180,E1 -8688.467,E2 -8688.467} C_VEL
LIN {X 0,Y 447.729,Z 772.965,A -85,B 0,C 180,E1 -8691.708,E2 -8691.708} C_VEL
LIN {X 0,Y 448.415,Z 778.079,A -85,B 0,C 180,E1 -8694.003,E2 -8694.003} C_VEL
LIN {X 0,Y 448.068,Z 784.538,A -85,B 0,C 180,E1 -8696.703,E2 -8696.703} C_VEL
LIN {X 0,Y 447.544,Z 792.292,A -85,B 0,C 180,E1 -8699.834,E2 -8699.834} C_VEL
LIN {X 0,Y 447.102,Z 800.068,A -85,B 0,C 180,E1 -8702.88,E2 -8702.88} C_VEL
LIN {X 0,Y 446.711,Z 807.874,A -85,B 0,C 180,E1 -8705.855,E2 -8705.855} C_VEL
LIN {X 0,Y 446.332,Z 816.999,A -85,B 0,C 180,E1 -8709.25,E2 -8709.25} C_VEL
LIN {X 0,Y 446.033,Z 824.837,A -85,B 0,C 180,E1 -8712.106,E2 -8712.106} C_VEL
LIN {X 0,Y 445.897,Z 829.819,A -85,B 0,C 180,E1 -8713.891,E2 -8713.891} C_VEL
LIN {X 0,Y 447.93,Z 843.636,A -85,B 0,C 180,E1 -8714.363,E2 -8714.363} C_VEL
LIN {X 0,Y 449.213,Z 853.188,A -85,B 0,C 180,E1 -8714.808,E2 -8714.808} C_VEL
LIN {X 0,Y 448.61,Z 865.683,A -85,B 0,C 180,E1 -8715.483,E2 -8715.483} C_VEL
LIN {X 0,Y 447.957,Z 878.282,A -85,B 0,C 180,E1 -8716.389,E2 -8716.389} C_VEL
LIN {X 0,Y 447.374,Z 889.48,A -85,B 0,C 180,E1 -8717.41,E2 -8717.41} C_VEL
LIN {X 0,Y 446.897,Z 898.552,A -85,B 0,C 180,E1 -8718.433,E2 -8718.433} C_VEL
LIN {X 0,Y 446.354,Z 908.391,A -85,B 0,C 180,E1 -8719.797,E2 -8719.797} C_VEL
LIN {X 0,Y 445.965,Z 916.295,A -85,B 0,C 180,E1 -8721.161,E2 -8721.161} C_VEL
LIN {X 0,Y 445.686,Z 923.528,A -85,B 0,C 180,E1 -8722.753,E2 -8722.753} C_VEL
LIN {X 0,Y 445.514,Z 928.716,A -85,B 0,C 180,E1 -8724.229,E2 -8724.229} C_VEL
LIN {X 0,Y 445.429,Z 932.037,A -85,B 0,C 180,E1 -8725.475,E2 -8725.475} C_VEL
LIN {X 0,Y 445.426,Z 933.937,A -85,B 0,C 180,E1 -8726.381,E2 -8726.381} C_VEL
LIN {X 0,Y 445.428,Z 935.363,A -85,B 0,C 180,E1 -8727.287,E2 -8727.287} C_VEL
LIN {X 0,Y 445.439,Z 936.365,A -85,B 0,C 180,E1 -8728.192,E2 -8728.192} C_VEL
LIN {X 0,Y 445.427,Z 936.967,A -85,B 0,C 180,E1 -8729.096,E2 -8729.096} C_VEL
LIN {X 0,Y 445.4,Z 937.166,A -85,B 0,C 180,E1 -8730,E2 -8730} C_VEL
LIN {X 0,Y 445.427,Z 936.921,A -85,B 0,C 180,E1 -8730.904,E2 -8730.904} C_VEL
LIN {X 0,Y 445.439,Z 936.265,A -85,B 0,C 180,E1 -8731.808,E2 -8731.808} C_VEL
LIN {X 0,Y 445.431,Z 935.206,A -85,B 0,C 180,E1 -8732.713,E2 -8732.713} C_VEL
LIN {X 0,Y 445.455,Z 933.73,A -85,B 0,C 180,E1 -8733.618,E2 -8733.618} C_VEL
LIN {X 0,Y 445.505,Z 930.65,A -85,B 0,C 180,E1 -8734.978,E2 -8734.978} C_VEL
LIN {X 0,Y 445.571,Z 926.162,A -85,B 0,C 180,E1 -8736.431,E2 -8736.431} C_VEL
LIN {X 0,Y 445.755,Z 920.103,A -85,B 0,C 180,E1 -8737.93,E2 -8737.93} C_VEL
LIN {X 0,Y 446.08,Z 913.155,A -85,B 0,C 180,E1 -8739.293,E2 -8739.293} C_VEL
LIN {X 0,Y 446.449,Z 904.528,A -85,B 0,C 180,E1 -8740.659,E2 -8740.659} C_VEL
LIN {X 0,Y 446.98,Z 895.674,A -85,B 0,C 180,E1 -8741.795,E2 -8741.795} C_VEL
LIN {X 0,Y 447.527,Z 885.334,A -85,B 0,C 180,E1 -8742.882,E2 -8742.882} C_VEL
LIN {X 0,Y 448.052,Z 874.115,A -85,B 0,C 180,E1 -8743.84,E2 -8743.84} C_VEL
LIN {X 0,Y 448.665,Z 862.328,A -85,B 0,C 180,E1 -8744.631,E2 -8744.631} C_VEL
LIN {X 0,Y 448.979,Z 851.685,A -85,B 0,C 180,E1 -8745.2,E2 -8745.2} C_VEL
LIN {X 0,Y 447.199,Z 838.034,A -85,B 0,C 180,E1 -8745.818,E2 -8745.818} C_VEL
LIN {X 0,Y 445.885,Z 828.009,A -85,B 0,C 180,E1 -8746.151,E2 -8746.151} C_VEL
LIN {X 0,Y 446.047,Z 818.938,A -85,B 0,C 180,E1 -8749.322,E2 -8749.322} C_VEL
LIN {X 0,Y 446.372,Z 809.589,A -85,B 0,C 180,E1 -8752.69,E2 -8752.69} C_VEL
LIN {X 0,Y 446.694,Z 801.732,A -85,B 0,C 180,E1 -8755.637,E2 -8755.637} C_VEL
LIN {X 0,Y 447.082,Z 794.076,A -85,B 0,C 180,E1 -8758.682,E2 -8758.682} C_VEL
LIN {X 0,Y 447.727,Z 785.832,A -85,B 0,C 180,E1 -8762.256,E2 -8762.256} C_VEL
LIN {X 0,Y 448.141,Z 781.452,A -85,B 0,C 180,E1 -8764.373,E2 -8764.373} C_VEL
LIN {X 0,Y 448.334,Z 777.448,A -85,B 0,C 180,E1 -8766.561,E2 -8766.561} C_VEL
LIN {X 0,Y 447.818,Z 773.958,A -85,B 0,C 180,E1 -8768.885,E2 -8768.885} C_VEL
LIN {X 0,Y 447.395,Z 771.108,A -85,B 0,C 180,E1 -8771.282,E2 -8771.282} C_VEL
LIN {X 0,Y 446.992,Z 769.001,A -85,B 0,C 180,E1 -8773.774,E2 -8773.774} C_VEL
LIN {X 0,Y 446.724,Z 767.679,A -85,B 0,C 180,E1 -8776.36,E2 -8776.36} C_VEL
LIN {X 0,Y 446.645,Z 767.173,A -85,B 0,C 180,E1 -8779.051,E2 -8779.051} C_VEL
LIN {X 0,Y 446.676,Z 767.47,A -85,B 0,C 180,E1 -8782.147,E2 -8782.147} C_VEL
LIN {X 0,Y 446.692,Z 768.351,A -85,B 0,C 180,E1 -8784.899,E2 -8784.899} C_VEL
LIN {X 0,Y 446.521,Z 769.686,A -85,B 0,C 180,E1 -8787.646,E2 -8787.646} C_VEL
LIN {X 0,Y 446.271,Z 771.58,A -85,B 0,C 180,E1 -8790.777,E2 -8790.777} C_VEL
LIN {X 0,Y 446.087,Z 773.748,A -85,B 0,C 180,E1 -8793.9,E2 -8793.9} C_VEL
LIN {X 0,Y 445.956,Z 775.946,A -85,B 0,C 180,E1 -8796.796,E2 -8796.796} C_VEL
LIN {X 0,Y 445.842,Z 778.315,A -85,B 0,C 180,E1 -8799.708,E2 -8799.708} C_VEL
LIN {X 0,Y 445.705,Z 780.78,A -85,B 0,C 180,E1 -8802.566,E2 -8802.566} C_VEL
LIN {X 0,Y 445.768,Z 782.251,A -85,B 0,C 180,E1 -8804.003,E2 -8804.003} C_VEL
LIN {X 0,Y 448.924,Z 794.568,A -85,B 0,C 180,E1 -8804.565,E2 -8804.565} C_VEL
LIN {X 0,Y 449.576,Z 799.671,A -85,B 0,C 180,E1 -8804.82,E2 -8804.82} C_VEL
LIN {X 0,Y 449.092,Z 812.21,A -85,B 0,C 180,E1 -8805.499,E2 -8805.499} C_VEL
LIN {X 0,Y 448.581,Z 823.004,A -85,B 0,C 180,E1 -8806.256,E2 -8806.256} C_VEL
LIN {X 0,Y 448.053,Z 833.757,A -85,B 0,C 180,E1 -8807.207,E2 -8807.207} C_VEL
LIN {X 0,Y 447.426,Z 843.117,A -85,B 0,C 180,E1 -8808.217,E2 -8808.217} C_VEL
LIN {X 0,Y 447.012,Z 851.772,A -85,B 0,C 180,E1 -8809.353,E2 -8809.353} C_VEL
LIN {X 0,Y 446.498,Z 860.197,A -85,B 0,C 180,E1 -8810.715,E2 -8810.715} C_VEL
LIN {X 0,Y 446.174,Z 865.934,A -85,B 0,C 180,E1 -8811.849,E2 -8811.849} C_VEL
LIN {X 0,Y 445.921,Z 871.392,A -85,B 0,C 180,E1 -8813.18,E2 -8813.18} C_VEL
LIN {X 0,Y 445.644,Z 875.865,A -85,B 0,C 180,E1 -8814.57,E2 -8814.57} C_VEL
LIN {X 0,Y 445.634,Z 878.153,A -85,B 0,C 180,E1 -8815.476,E2 -8815.476} C_VEL
LIN {X 0,Y 445.587,Z 880.015,A -85,B 0,C 180,E1 -8816.382,E2 -8816.382} C_VEL
LIN {X 0,Y 445.505,Z 881.43,A -85,B 0,C 180,E1 -8817.286,E2 -8817.286} C_VEL
LIN {X 0,Y 445.509,Z 882.41,A -85,B 0,C 180,E1 -8818.191,E2 -8818.191} C_VEL
LIN {X 0,Y 445.4,Z 883.217,A -85,B 0,C 180,E1 -8819.999,E2 -8819.999} C_VEL
LIN {X 0,Y 445.427,Z 882.995,A -85,B 0,C 180,E1 -8820.903,E2 -8820.903} C_VEL
LIN {X 0,Y 445.504,Z 882.364,A -85,B 0,C 180,E1 -8821.807,E2 -8821.807} C_VEL
LIN {X 0,Y 445.473,Z 881.352,A -85,B 0,C 180,E1 -8822.712,E2 -8822.712} C_VEL
LIN {X 0,Y 445.577,Z 879.934,A -85,B 0,C 180,E1 -8823.616,E2 -8823.616} C_VEL
LIN {X 0,Y 445.555,Z 876.975,A -85,B 0,C 180,E1 -8824.976,E2 -8824.976} C_VEL
LIN {X 0,Y 445.843,Z 872.961,A -85,B 0,C 180,E1 -8826.334,E2 -8826.334} C_VEL
LIN {X 0,Y 446.025,Z 866.79,A -85,B 0,C 180,E1 -8827.924,E2 -8827.924} C_VEL
LIN {X 0,Y 446.413,Z 860.048,A -85,B 0,C 180,E1 -8829.285,E2 -8829.285} C_VEL
LIN {X 0,Y 446.893,Z 851.685,A -85,B 0,C 180,E1 -8830.648,E2 -8830.648} C_VEL
LIN {X 0,Y 447.363,Z 843.076,A -85,B 0,C 180,E1 -8831.783,E2 -8831.783} C_VEL
LIN {X 0,Y 447.948,Z 832.967,A -85,B 0,C 180,E1 -8832.871,E2 -8832.871} C_VEL
LIN {X 0,Y 448.447,Z 822.039,A -85,B 0,C 180,E1 -8833.826,E2 -8833.826} C_VEL
LIN {X 0,Y 448.975,Z 810.546,A -85,B 0,C 180,E1 -8834.619,E2 -8834.619} C_VEL
LIN {X 0,Y 449.406,Z 798.805,A -85,B 0,C 180,E1 -8835.242,E2 -8835.242} C_VEL
LIN {X 0,Y 447.665,Z 789.093,A -85,B 0,C 180,E1 -8835.707,E2 -8835.707} C_VEL
LIN {X 0,Y 445.535,Z 779.918,A -85,B 0,C 180,E1 -8836.096,E2 -8836.096} C_VEL
LIN {X 0,Y 445.535,Z 776.521,A -85,B 0,C 180,E1 -8839.344,E2 -8839.344} C_VEL
LIN {X 0,Y 445.576,Z 773.523,A -85,B 0,C 180,E1 -8842.243,E2 -8842.243} C_VEL
LIN {X 0,Y 445.651,Z 770.513,A -85,B 0,C 180,E1 -8845.2,E2 -8845.2} C_VEL
LIN {X 0,Y 445.685,Z 767.485,A -85,B 0,C 180,E1 -8848.232,E2 -8848.232} C_VEL
LIN {X 0,Y 445.761,Z 765.962,A -85,B 0,C 180,E1 -8849.871,E2 -8849.871} C_VEL
LIN {X 0,Y 446.065,Z 765.925,A -85,B 0,C 180,E1 -8852.389,E2 -8852.389} C_VEL
LIN {X 0,Y 446.343,Z 765.886,A -85,B 0,C 180,E1 -8855.632,E2 -8855.632} C_VEL
LIN {X 0,Y 446.439,Z 765.877,A -85,B 0,C 180,E1 -8859.026,E2 -8859.026} C_VEL
LIN {X 0,Y 446.43,Z 765.874,A -85,B 0,C 180,E1 -8862.276,E2 -8862.276} C_VEL
LIN {X 0,Y 446.448,Z 765.876,A -85,B 0,C 180,E1 -8865.102,E2 -8865.102} C_VEL
LIN {X 0,Y 446.422,Z 765.875,A -85,B 0,C 180,E1 -8868.608,E2 -8868.608} C_VEL
LIN {X 0,Y 446.435,Z 765.875,A -85,B 0,C 180,E1 -8870.972,E2 -8870.972} C_VEL
LIN {X 0,Y 446.411,Z 765.876,A -85,B 0,C 180,E1 -8874.373,E2 -8874.373} C_VEL
LIN {X 0,Y 446.412,Z 765.878,A -85,B 0,C 180,E1 -8877.637,E2 -8877.637} C_VEL
LIN {X 0,Y 446.429,Z 765.873,A -85,B 0,C 180,E1 -8880.789,E2 -8880.789} C_VEL
LIN {X 0,Y 446.43,Z 765.875,A -85,B 0,C 180,E1 -8883.845,E2 -8883.845} C_VEL
LIN {X 0,Y 446.415,Z 765.875,A -85,B 0,C 180,E1 -8886.822,E2 -8886.822} C_VEL
LIN {X 0,Y 446.434,Z 765.877,A -85,B 0,C 180,E1 -8889.737,E2 -8889.737} C_VEL
LIN {X 0,Y 446.445,Z 765.871,A -85,B 0,C 180,E1 -8892.596,E2 -8892.596} C_VEL
LIN {X 0,Y 446.459,Z 765.872,A -85,B 0,C 180,E1 -8895.412,E2 -8895.412} C_VEL
LIN {X 0,Y 446.506,Z 765.865,A -85,B 0,C 180,E1 -8898.193,E2 -8898.193} C_VEL
LIN {X 0,Y 446.515,Z 765.861,A -85,B 0,C 180,E1 -8900.944,E2 -8900.944} C_VEL
LIN {X 0,Y 446.561,Z 765.855,A -85,B 0,C 180,E1 -8903.01,E2 -8903.01} C_VEL
LIN {X 0,Y 445.869,Z 765.947,A -85,B 0,C 180,E1 -8903.762,E2 -8903.762} C_VEL
LIN {X 0,Y 442.909,Z 766.311,A -85,B 0,C 180,E1 -8904.983,E2 -8904.983} C_VEL
LIN {X 0,Y 440.477,Z 766.62,A -85,B 0,C 180,E1 -8905.968,E2 -8905.968} C_VEL
LIN {X 0,Y 439.537,Z 766.731,A -85,B 0,C 180,E1 -8906.73,E2 -8906.73} C_VEL
LIN {X 0,Y 439.516,Z 766.732,A -85,B 0,C 180,E1 -8906.988,E2 -8906.988} C_VEL
LIN {X 0,Y 439.658,Z 766.723,A -85,B 0,C 180,E1 -8910,E2 -8910} C_VEL
LIN {X 0,Y 439.59,Z 766.724,A -85,B 0,C 180,E1 -8912.749,E2 -8912.749} C_VEL
LIN {X 0,Y 439.546,Z 766.733,A -85,B 0,C 180,E1 -8916.426,E2 -8916.426} C_VEL
LIN {X 0,Y 439.462,Z 766.739,A -85,B 0,C 180,E1 -8919.202,E2 -8919.202} C_VEL
LIN {X 0,Y 439.456,Z 766.741,A -85,B 0,C 180,E1 -8922.938,E2 -8922.938} C_VEL
LIN {X 0,Y 439.436,Z 766.75,A -85,B 0,C 180,E1 -8926.348,E2 -8926.348} C_VEL
LIN {X 0,Y 439.392,Z 766.749,A -85,B 0,C 180,E1 -8929.627,E2 -8929.627} C_VEL
LIN {X 0,Y 439.354,Z 766.759,A -85,B 0,C 180,E1 -8932.576,E2 -8932.576} C_VEL
LIN {X 0,Y 439.363,Z 766.753,A -85,B 0,C 180,E1 -8935.588,E2 -8935.588} C_VEL
LIN {X 0,Y 439.388,Z 766.756,A -85,B 0,C 180,E1 -8938.676,E2 -8938.676} C_VEL
LIN {X 0,Y 439.36,Z 766.754,A -85,B 0,C 180,E1 -8942.031,E2 -8942.031} C_VEL
LIN {X 0,Y 439.385,Z 766.751,A -85,B 0,C 180,E1 -8945.341,E2 -8945.341} C_VEL
LIN {X 0,Y 439.37,Z 766.756,A -85,B 0,C 180,E1 -8948.596,E2 -8948.596} C_VEL
LIN {X 0,Y 439.382,Z 766.753,A -85,B 0,C 180,E1 -8951.258,E2 -8951.258} C_VEL
LIN {X 0,Y 439.394,Z 766.753,A -85,B 0,C 180,E1 -8954.73,E2 -8954.73} C_VEL
LIN {X 0,Y 439.391,Z 766.751,A -85,B 0,C 180,E1 -8957.797,E2 -8957.797} C_VEL
LIN {X 0,Y 439.421,Z 766.748,A -85,B 0,C 180,E1 -8960.228,E2 -8960.228} C_VEL
LIN {X 0,Y 439.347,Z 766.757,A -85,B 0,C 180,E1 -8963.712,E2 -8963.712} C_VEL
LIN {X 0,Y 439.184,Z 766.779,A -85,B 0,C 180,E1 -8966.318,E2 -8966.318} C_VEL
LIN {X 0,Y 438.832,Z 766.825,A -85,B 0,C 180,E1 -8969.172,E2 -8969.172} C_VEL
LIN {X 0,Y 438.528,Z 767.109,A -85,B 0,C 180,E1 -8971.818,E2 -8971.818} C_VEL
LIN {X 0,Y 438.554,Z 769.871,A -85,B 0,C 180,E1 -8974.363,E2 -8974.363} C_VEL
LIN {X 0,Y 438.47,Z 773.135,A -85,B 0,C 180,E1 -8977.377,E2 -8977.377} C_VEL
LIN {X 0,Y 438.46,Z 776.328,A -85,B 0,C 180,E1 -8980.331,E2 -8980.331} C_VEL
LIN {X 0,Y 438.44,Z 780.213,A -85,B 0,C 180,E1 -8983.792,E2 -8983.792} C_VEL
LIN {X 0,Y 441.547,Z 793.671,A -85,B 0,C 180,E1 -8984.361,E2 -8984.361} C_VEL
LIN {X 0,Y 442.495,Z 800.139,A -85,B 0,C 180,E1 -8984.691,E2 -8984.691} C_VEL
LIN {X 0,Y 441.989,Z 812.491,A -85,B 0,C 180,E1 -8985.38,E2 -8985.38} C_VEL
LIN {X 0,Y 441.419,Z 824.048,A -85,B 0,C 180,E1 -8986.218,E2 -8986.218} C_VEL
LIN {X 0,Y 440.914,Z 834.975,A -85,B 0,C 180,E1 -8987.224,E2 -8987.224} C_VEL
LIN {X 0,Y 440.289,Z 844.203,A -85,B 0,C 180,E1 -8988.258,E2 -8988.258} C_VEL
LIN {X 0,Y 439.835,Z 852.682,A -85,B 0,C 180,E1 -8989.412,E2 -8989.412} C_VEL
LIN {X 0,Y 439.356,Z 860.919,A -85,B 0,C 180,E1 -8990.796,E2 -8990.796} C_VEL
LIN {X 0,Y 438.945,Z 867.557,A -85,B 0,C 180,E1 -8992.179,E2 -8992.179} C_VEL
LIN {X 0,Y 438.77,Z 872.851,A -85,B 0,C 180,E1 -8993.563,E2 -8993.563} C_VEL
LIN {X 0,Y 438.498,Z 876.973,A -85,B 0,C 180,E1 -8994.944,E2 -8994.944} C_VEL
LIN {X 0,Y 438.511,Z 880.021,A -85,B 0,C 180,E1 -8996.325,E2 -8996.325} C_VEL
LIN {X 0,Y 438.395,Z 881.525,A -85,B 0,C 180,E1 -8997.244,E2 -8997.244} C_VEL
LIN {X 0,Y 438.413,Z 882.575,A -85,B 0,C 180,E1 -8998.164,E2 -8998.164} C_VEL
LIN {X 0,Y 438.338,Z 883.526,A -85,B 0,C 180,E1 -9000.001,E2 -9000.001} C_VEL
LIN {X 0,Y 438.367,Z 883.364,A -85,B 0,C 180,E1 -9000.92,E2 -9000.92} C_VEL
LIN {X 0,Y 438.431,Z 882.8,A -85,B 0,C 180,E1 -9001.838,E2 -9001.838} C_VEL
LIN {X 0,Y 438.414,Z 881.855,A -85,B 0,C 180,E1 -9002.757,E2 -9002.757} C_VEL
LIN {X 0,Y 438.523,Z 880.486,A -85,B 0,C 180,E1 -9003.676,E2 -9003.676} C_VEL
LIN {X 0,Y 438.53,Z 877.614,A -85,B 0,C 180,E1 -9005.058,E2 -9005.058} C_VEL
LIN {X 0,Y 438.837,Z 873.669,A -85,B 0,C 180,E1 -9006.438,E2 -9006.438} C_VEL
LIN {X 0,Y 438.998,Z 868.56,A -85,B 0,C 180,E1 -9007.822,E2 -9007.822} C_VEL
LIN {X 0,Y 439.384,Z 862.137,A -85,B 0,C 180,E1 -9009.205,E2 -9009.205} C_VEL
LIN {X 0,Y 439.908,Z 854.162,A -85,B 0,C 180,E1 -9010.588,E2 -9010.588} C_VEL
LIN {X 0,Y 440.38,Z 845.981,A -85,B 0,C 180,E1 -9011.741,E2 -9011.741} C_VEL
LIN {X 0,Y 441.048,Z 835.921,A -85,B 0,C 180,E1 -9012.891,E2 -9012.891} C_VEL
LIN {X 0,Y 441.547,Z 824.741,A -85,B 0,C 180,E1 -9013.931,E2 -9013.931} C_VEL
LIN {X 0,Y 442.245,Z 811.908,A -85,B 0,C 180,E1 -9014.849,E2 -9014.849} C_VEL
LIN {X 0,Y 442.718,Z 800.475,A -85,B 0,C 180,E1 -9015.48,E2 -9015.48} C_VEL
LIN {X 0,Y 441.198,Z 791.963,A -85,B 0,C 180,E1 -9015.922,E2 -9015.922} C_VEL
LIN {X 0,Y 438.606,Z 781.972,A -85,B 0,C 180,E1 -9016.386,E2 -9016.386} C_VEL
LIN {X 0,Y 438.615,Z 778.44,A -85,B 0,C 180,E1 -9019.664,E2 -9019.664} C_VEL
LIN {X 0,Y 438.644,Z 775.179,A -85,B 0,C 180,E1 -9022.615,E2 -9022.615} C_VEL
LIN {X 0,Y 438.663,Z 772.885,A -85,B 0,C 180,E1 -9024.618,E2 -9024.618} C_VEL
LIN {X 0,Y 438.679,Z 769.309,A -85,B 0,C 180,E1 -9027.685,E2 -9027.685} C_VEL
LIN {X 0,Y 438.696,Z 766.844,A -85,B 0,C 180,E1 -9029.778,E2 -9029.778} C_VEL
LIN {X 0,Y 439.104,Z 766.792,A -85,B 0,C 180,E1 -9032.969,E2 -9032.969} C_VEL
LIN {X 0,Y 439.316,Z 766.765,A -85,B 0,C 180,E1 -9035.325,E2 -9035.325} C_VEL
LIN {X 0,Y 439.373,Z 766.755,A -85,B 0,C 180,E1 -9038.597,E2 -9038.597} C_VEL
LIN {X 0,Y 439.386,Z 766.756,A -85,B 0,C 180,E1 -9041.256,E2 -9041.256} C_VEL
LIN {X 0,Y 439.405,Z 766.754,A -85,B 0,C 180,E1 -9044.73,E2 -9044.73} C_VEL
LIN {X 0,Y 439.443,Z 766.944,A -85,B 0,C 180,E1 -9048.171,E2 -9048.171} C_VEL
LIN {X 0,Y 440.706,Z 773.953,A -85,B 0,C 180,E1 -9051.542,E2 -9051.542} C_VEL
LIN {X 0,Y 441.423,Z 779.141,A -85,B 0,C 180,E1 -9053.908,E2 -9053.908} C_VEL
LIN {X 0,Y 441.086,Z 785.593,A -85,B 0,C 180,E1 -9056.653,E2 -9056.653} C_VEL
LIN {X 0,Y 440.516,Z 793.538,A -85,B 0,C 180,E1 -9059.913,E2 -9059.913} C_VEL
LIN {X 0,Y 440.054,Z 801.104,A -85,B 0,C 180,E1 -9062.924,E2 -9062.924} C_VEL
LIN {X 0,Y 439.63,Z 809.166,A -85,B 0,C 180,E1 -9066.048,E2 -9066.048} C_VEL
LIN {X 0,Y 439.253,Z 817.992,A -85,B 0,C 180,E1 -9069.39,E2 -9069.39} C_VEL
LIN {X 0,Y 438.887,Z 827.106,A -85,B 0,C 180,E1 -9072.768,E2 -9072.768} C_VEL
LIN {X 0,Y 438.824,Z 829.47,A -85,B 0,C 180,E1 -9073.635,E2 -9073.635} C_VEL
LIN {X 0,Y 440.922,Z 843.779,A -85,B 0,C 180,E1 -9074.145,E2 -9074.145} C_VEL
LIN {X 0,Y 442.244,Z 854.842,A -85,B 0,C 180,E1 -9074.681,E2 -9074.681} C_VEL
LIN {X 0,Y 441.601,Z 866.744,A -85,B 0,C 180,E1 -9075.366,E2 -9075.366} C_VEL
LIN {X 0,Y 440.951,Z 878.894,A -85,B 0,C 180,E1 -9076.272,E2 -9076.272} C_VEL
LIN {X 0,Y 440.339,Z 889.974,A -85,B 0,C 180,E1 -9077.323,E2 -9077.323} C_VEL
LIN {X 0,Y 439.78,Z 899.796,A -85,B 0,C 180,E1 -9078.477,E2 -9078.477} C_VEL
LIN {X 0,Y 439.308,Z 907.873,A -85,B 0,C 180,E1 -9079.632,E2 -9079.632} C_VEL
LIN {X 0,Y 438.897,Z 915.809,A -85,B 0,C 180,E1 -9081.018,E2 -9081.018} C_VEL
LIN {X 0,Y 438.659,Z 921.193,A -85,B 0,C 180,E1 -9082.173,E2 -9082.173} C_VEL
LIN {X 0,Y 438.508,Z 926.449,A -85,B 0,C 180,E1 -9083.558,E2 -9083.558} C_VEL
LIN {X 0,Y 438.435,Z 930.516,A -85,B 0,C 180,E1 -9084.942,E2 -9084.942} C_VEL
LIN {X 0,Y 438.329,Z 933.503,A -85,B 0,C 180,E1 -9086.323,E2 -9086.323} C_VEL
LIN {X 0,Y 438.357,Z 934.935,A -85,B 0,C 180,E1 -9087.243,E2 -9087.243} C_VEL
LIN {X 0,Y 438.354,Z 935.938,A -85,B 0,C 180,E1 -9088.162,E2 -9088.162} C_VEL
LIN {X 0,Y 438.366,Z 936.541,A -85,B 0,C 180,E1 -9089.081,E2 -9089.081} C_VEL
LIN {X 0,Y 438.338,Z 936.738,A -85,B 0,C 180,E1 -9090,E2 -9090} C_VEL
LIN {X 0,Y 438.366,Z 936.489,A -85,B 0,C 180,E1 -9090.919,E2 -9090.919} C_VEL
LIN {X 0,Y 438.354,Z 935.829,A -85,B 0,C 180,E1 -9091.838,E2 -9091.838} C_VEL
LIN {X 0,Y 438.362,Z 934.767,A -85,B 0,C 180,E1 -9092.757,E2 -9092.757} C_VEL
LIN {X 0,Y 438.356,Z 933.281,A -85,B 0,C 180,E1 -9093.677,E2 -9093.677} C_VEL
LIN {X 0,Y 438.44,Z 930.191,A -85,B 0,C 180,E1 -9095.058,E2 -9095.058} C_VEL
LIN {X 0,Y 438.474,Z 926.013,A -85,B 0,C 180,E1 -9096.442,E2 -9096.442} C_VEL
LIN {X 0,Y 438.703,Z 919.603,A -85,B 0,C 180,E1 -9098.058,E2 -9098.058} C_VEL
LIN {X 0,Y 439.017,Z 912.624,A -85,B 0,C 180,E1 -9099.444,E2 -9099.444} C_VEL
LIN {X 0,Y 439.428,Z 903.969,A -85,B 0,C 180,E1 -9100.832,E2 -9100.832} C_VEL
LIN {X 0,Y 440.086,Z 893.12,A -85,B 0,C 180,E1 -9102.216,E2 -9102.216} C_VEL
LIN {X 0,Y 440.622,Z 882.928,A -85,B 0,C 180,E1 -9103.271,E2 -9103.271} C_VEL
LIN {X 0,Y 441.2,Z 872.105,A -85,B 0,C 180,E1 -9104.177,E2 -9104.177} C_VEL
